   STATUS[376].EXT.AckRequired := FALSE;
   STATUS[376].EXT.Maintanence := FALSE;
   STATUS[376].EXT.Operation := FALSE;
   STATUS[376].EXT.Forced := FALSE;
   STATUS[376].EXT.BIT29 := FALSE;
   STATUS[376].EXT.BIT30 := FALSE;
   STATUS[376].EXT.BIT31 := FALSE;
   STATUS[376].EXT.ModeBit1 := FALSE;
   STATUS[376].EXT.ModeBit2 := FALSE;
   STATUS[376].EXT.ModeBit3 := FALSE;
   STATUS[376].EXT.BIT19 := FALSE;
   STATUS[376].EXT.BIT20 := FALSE;
   STATUS[376].EXT.AlarmSuppressed := FALSE;
   STATUS[376].EXT.AlarmPresent := FALSE;
   STATUS[376].EXT.AlarmFailUnAck := FALSE;
   STATUS[376].Status := 0;
   STATUS[376].TimeStamp := 16#0000;
   STATUS[377].EXT.AlarmWarnUnAck := FALSE;
   STATUS[377].EXT.AckRequired := FALSE;
   STATUS[377].EXT.Maintanence := FALSE;
   STATUS[377].EXT.Operation := FALSE;
   STATUS[377].EXT.Forced := FALSE;
   STATUS[377].EXT.BIT29 := FALSE;
   STATUS[377].EXT.BIT30 := FALSE;
   STATUS[377].EXT.BIT31 := FALSE;
   STATUS[377].EXT.ModeBit1 := FALSE;
   STATUS[377].EXT.ModeBit2 := FALSE;
   STATUS[377].EXT.ModeBit3 := FALSE;
   STATUS[377].EXT.BIT19 := FALSE;
   STATUS[377].EXT.BIT20 := FALSE;
   STATUS[377].EXT.AlarmSuppressed := FALSE;
   STATUS[377].EXT.AlarmPresent := FALSE;
   STATUS[377].EXT.AlarmFailUnAck := FALSE;
   STATUS[377].Status := 0;
   STATUS[377].TimeStamp := 16#0000;
   STATUS[378].EXT.AlarmWarnUnAck := FALSE;
   STATUS[378].EXT.AckRequired := FALSE;
   STATUS[378].EXT.Maintanence := FALSE;
   STATUS[378].EXT.Operation := FALSE;
   STATUS[378].EXT.Forced := FALSE;
   STATUS[378].EXT.BIT29 := FALSE;
   STATUS[378].EXT.BIT30 := FALSE;
   STATUS[378].EXT.BIT31 := FALSE;
   STATUS[378].EXT.ModeBit1 := FALSE;
   STATUS[378].EXT.ModeBit2 := FALSE;
   STATUS[378].EXT.ModeBit3 := FALSE;
   STATUS[378].EXT.BIT19 := FALSE;
   STATUS[378].EXT.BIT20 := FALSE;
   STATUS[378].EXT.AlarmSuppressed := FALSE;
   STATUS[378].EXT.AlarmPresent := FALSE;
   STATUS[378].EXT.AlarmFailUnAck := FALSE;
   STATUS[378].Status := 0;
   STATUS[378].TimeStamp := 16#0000;
   STATUS[379].EXT.AlarmWarnUnAck := FALSE;
   STATUS[379].EXT.AckRequired := FALSE;
   STATUS[379].EXT.Maintanence := FALSE;
   STATUS[379].EXT.Operation := FALSE;
   STATUS[379].EXT.Forced := FALSE;
   STATUS[379].EXT.BIT29 := FALSE;
   STATUS[379].EXT.BIT30 := FALSE;
   STATUS[379].EXT.BIT31 := FALSE;
   STATUS[379].EXT.ModeBit1 := FALSE;
   STATUS[379].EXT.ModeBit2 := FALSE;
   STATUS[379].EXT.ModeBit3 := FALSE;
   STATUS[379].EXT.BIT19 := FALSE;
   STATUS[379].EXT.BIT20 := FALSE;
   STATUS[379].EXT.AlarmSuppressed := FALSE;
   STATUS[379].EXT.AlarmPresent := FALSE;
   STATUS[379].EXT.AlarmFailUnAck := FALSE;
   STATUS[379].Status := 0;
   STATUS[379].TimeStamp := 16#0000;
   STATUS[380].EXT.AlarmWarnUnAck := FALSE;
   STATUS[380].EXT.AckRequired := FALSE;
   STATUS[380].EXT.Maintanence := FALSE;
   STATUS[380].EXT.Operation := FALSE;
   STATUS[380].EXT.Forced := FALSE;
   STATUS[380].EXT.BIT29 := FALSE;
   STATUS[380].EXT.BIT30 := FALSE;
   STATUS[380].EXT.BIT31 := FALSE;
   STATUS[380].EXT.ModeBit1 := FALSE;
   STATUS[380].EXT.ModeBit2 := FALSE;
   STATUS[380].EXT.ModeBit3 := FALSE;
   STATUS[380].EXT.BIT19 := FALSE;
   STATUS[380].EXT.BIT20 := FALSE;
   STATUS[380].EXT.AlarmSuppressed := FALSE;
   STATUS[380].EXT.AlarmPresent := FALSE;
   STATUS[380].EXT.AlarmFailUnAck := FALSE;
   STATUS[380].Status := 0;
   STATUS[380].TimeStamp := 16#0000;
   STATUS[381].EXT.AlarmWarnUnAck := FALSE;
   STATUS[381].EXT.AckRequired := FALSE;
   STATUS[381].EXT.Maintanence := FALSE;
   STATUS[381].EXT.Operation := FALSE;
   STATUS[381].EXT.Forced := FALSE;
   STATUS[381].EXT.BIT29 := FALSE;
   STATUS[381].EXT.BIT30 := FALSE;
   STATUS[381].EXT.BIT31 := FALSE;
   STATUS[381].EXT.ModeBit1 := FALSE;
   STATUS[381].EXT.ModeBit2 := FALSE;
   STATUS[381].EXT.ModeBit3 := FALSE;
   STATUS[381].EXT.BIT19 := FALSE;
   STATUS[381].EXT.BIT20 := FALSE;
   STATUS[381].EXT.AlarmSuppressed := FALSE;
   STATUS[381].EXT.AlarmPresent := FALSE;
   STATUS[381].EXT.AlarmFailUnAck := FALSE;
   STATUS[381].Status := 0;
   STATUS[381].TimeStamp := 16#0000;
   STATUS[382].EXT.AlarmWarnUnAck := FALSE;
   STATUS[382].EXT.AckRequired := FALSE;
   STATUS[382].EXT.Maintanence := FALSE;
   STATUS[382].EXT.Operation := FALSE;
   STATUS[382].EXT.Forced := FALSE;
   STATUS[382].EXT.BIT29 := FALSE;
   STATUS[382].EXT.BIT30 := FALSE;
   STATUS[382].EXT.BIT31 := FALSE;
   STATUS[382].EXT.ModeBit1 := FALSE;
   STATUS[382].EXT.ModeBit2 := FALSE;
   STATUS[382].EXT.ModeBit3 := FALSE;
   STATUS[382].EXT.BIT19 := FALSE;
   STATUS[382].EXT.BIT20 := FALSE;
   STATUS[382].EXT.AlarmSuppressed := FALSE;
   STATUS[382].EXT.AlarmPresent := FALSE;
   STATUS[382].EXT.AlarmFailUnAck := FALSE;
   STATUS[382].Status := 0;
   STATUS[382].TimeStamp := 16#0000;
   STATUS[383].EXT.AlarmWarnUnAck := FALSE;
   STATUS[383].EXT.AckRequired := FALSE;
   STATUS[383].EXT.Maintanence := FALSE;
   STATUS[383].EXT.Operation := FALSE;
   STATUS[383].EXT.Forced := FALSE;
   STATUS[383].EXT.BIT29 := FALSE;
   STATUS[383].EXT.BIT30 := FALSE;
   STATUS[383].EXT.BIT31 := FALSE;
   STATUS[383].EXT.ModeBit1 := FALSE;
   STATUS[383].EXT.ModeBit2 := FALSE;
   STATUS[383].EXT.ModeBit3 := FALSE;
   STATUS[383].EXT.BIT19 := FALSE;
   STATUS[383].EXT.BIT20 := FALSE;
   STATUS[383].EXT.AlarmSuppressed := FALSE;
   STATUS[383].EXT.AlarmPresent := FALSE;
   STATUS[383].EXT.AlarmFailUnAck := FALSE;
   STATUS[383].Status := 0;
   STATUS[383].TimeStamp := 16#0000;
   STATUS[384].EXT.AlarmWarnUnAck := FALSE;
   STATUS[384].EXT.AckRequired := FALSE;
   STATUS[384].EXT.Maintanence := FALSE;
   STATUS[384].EXT.Operation := FALSE;
   STATUS[384].EXT.Forced := FALSE;
   STATUS[384].EXT.BIT29 := FALSE;
   STATUS[384].EXT.BIT30 := FALSE;
   STATUS[384].EXT.BIT31 := FALSE;
   STATUS[384].EXT.ModeBit1 := FALSE;
   STATUS[384].EXT.ModeBit2 := FALSE;
   STATUS[384].EXT.ModeBit3 := FALSE;
   STATUS[384].EXT.BIT19 := FALSE;
   STATUS[384].EXT.BIT20 := FALSE;
   STATUS[384].EXT.AlarmSuppressed := FALSE;
   STATUS[384].EXT.AlarmPresent := FALSE;
   STATUS[384].EXT.AlarmFailUnAck := FALSE;
   STATUS[384].Status := 0;
   STATUS[384].TimeStamp := 16#0000;
   STATUS[385].EXT.AlarmWarnUnAck := FALSE;
   STATUS[385].EXT.AckRequired := FALSE;
   STATUS[385].EXT.Maintanence := FALSE;
   STATUS[385].EXT.Operation := FALSE;
   STATUS[385].EXT.Forced := FALSE;
   STATUS[385].EXT.BIT29 := FALSE;
   STATUS[385].EXT.BIT30 := FALSE;
   STATUS[385].EXT.BIT31 := FALSE;
   STATUS[385].EXT.ModeBit1 := FALSE;
   STATUS[385].EXT.ModeBit2 := FALSE;
   STATUS[385].EXT.ModeBit3 := FALSE;
   STATUS[385].EXT.BIT19 := FALSE;
   STATUS[385].EXT.BIT20 := FALSE;
   STATUS[385].EXT.AlarmSuppressed := FALSE;
   STATUS[385].EXT.AlarmPresent := FALSE;
   STATUS[385].EXT.AlarmFailUnAck := FALSE;
   STATUS[385].Status := 0;
   STATUS[385].TimeStamp := 16#0000;
   STATUS[386].EXT.AlarmWarnUnAck := FALSE;
   STATUS[386].EXT.AckRequired := FALSE;
   STATUS[386].EXT.Maintanence := FALSE;
   STATUS[386].EXT.Operation := FALSE;
   STATUS[386].EXT.Forced := FALSE;
   STATUS[386].EXT.BIT29 := FALSE;
   STATUS[386].EXT.BIT30 := FALSE;
   STATUS[386].EXT.BIT31 := FALSE;
   STATUS[386].EXT.ModeBit1 := FALSE;
   STATUS[386].EXT.ModeBit2 := FALSE;
   STATUS[386].EXT.ModeBit3 := FALSE;
   STATUS[386].EXT.BIT19 := FALSE;
   STATUS[386].EXT.BIT20 := FALSE;
   STATUS[386].EXT.AlarmSuppressed := FALSE;
   STATUS[386].EXT.AlarmPresent := FALSE;
   STATUS[386].EXT.AlarmFailUnAck := FALSE;
   STATUS[386].Status := 0;
   STATUS[386].TimeStamp := 16#0000;
   STATUS[387].EXT.AlarmWarnUnAck := FALSE;
   STATUS[387].EXT.AckRequired := FALSE;
   STATUS[387].EXT.Maintanence := FALSE;
   STATUS[387].EXT.Operation := FALSE;
   STATUS[387].EXT.Forced := FALSE;
   STATUS[387].EXT.BIT29 := FALSE;
   STATUS[387].EXT.BIT30 := FALSE;
   STATUS[387].EXT.BIT31 := FALSE;
   STATUS[387].EXT.ModeBit1 := FALSE;
   STATUS[387].EXT.ModeBit2 := FALSE;
   STATUS[387].EXT.ModeBit3 := FALSE;
   STATUS[387].EXT.BIT19 := FALSE;
   STATUS[387].EXT.BIT20 := FALSE;
   STATUS[387].EXT.AlarmSuppressed := FALSE;
   STATUS[387].EXT.AlarmPresent := FALSE;
   STATUS[387].EXT.AlarmFailUnAck := FALSE;
   STATUS[387].Status := 0;
   STATUS[387].TimeStamp := 16#0000;
   STATUS[388].EXT.AlarmWarnUnAck := FALSE;
   STATUS[388].EXT.AckRequired := FALSE;
   STATUS[388].EXT.Maintanence := FALSE;
   STATUS[388].EXT.Operation := FALSE;
   STATUS[388].EXT.Forced := FALSE;
   STATUS[388].EXT.BIT29 := FALSE;
   STATUS[388].EXT.BIT30 := FALSE;
   STATUS[388].EXT.BIT31 := FALSE;
   STATUS[388].EXT.ModeBit1 := FALSE;
   STATUS[388].EXT.ModeBit2 := FALSE;
   STATUS[388].EXT.ModeBit3 := FALSE;
   STATUS[388].EXT.BIT19 := FALSE;
   STATUS[388].EXT.BIT20 := FALSE;
   STATUS[388].EXT.AlarmSuppressed := FALSE;
   STATUS[388].EXT.AlarmPresent := FALSE;
   STATUS[388].EXT.AlarmFailUnAck := FALSE;
   STATUS[388].Status := 0;
   STATUS[388].TimeStamp := 16#0000;
   STATUS[389].EXT.AlarmWarnUnAck := FALSE;
   STATUS[389].EXT.AckRequired := FALSE;
   STATUS[389].EXT.Maintanence := FALSE;
   STATUS[389].EXT.Operation := FALSE;
   STATUS[389].EXT.Forced := FALSE;
   STATUS[389].EXT.BIT29 := FALSE;
   STATUS[389].EXT.BIT30 := FALSE;
   STATUS[389].EXT.BIT31 := FALSE;
   STATUS[389].EXT.ModeBit1 := FALSE;
   STATUS[389].EXT.ModeBit2 := FALSE;
   STATUS[389].EXT.ModeBit3 := FALSE;
   STATUS[389].EXT.BIT19 := FALSE;
   STATUS[389].EXT.BIT20 := FALSE;
   STATUS[389].EXT.AlarmSuppressed := FALSE;
   STATUS[389].EXT.AlarmPresent := FALSE;
   STATUS[389].EXT.AlarmFailUnAck := FALSE;
   STATUS[389].Status := 0;
   STATUS[389].TimeStamp := 16#0000;
   STATUS[390].EXT.AlarmWarnUnAck := FALSE;
   STATUS[390].EXT.AckRequired := FALSE;
   STATUS[390].EXT.Maintanence := FALSE;
   STATUS[390].EXT.Operation := FALSE;
   STATUS[390].EXT.Forced := FALSE;
   STATUS[390].EXT.BIT29 := FALSE;
   STATUS[390].EXT.BIT30 := FALSE;
   STATUS[390].EXT.BIT31 := FALSE;
   STATUS[390].EXT.ModeBit1 := FALSE;
   STATUS[390].EXT.ModeBit2 := FALSE;
   STATUS[390].EXT.ModeBit3 := FALSE;
   STATUS[390].EXT.BIT19 := FALSE;
   STATUS[390].EXT.BIT20 := FALSE;
   STATUS[390].EXT.AlarmSuppressed := FALSE;
   STATUS[390].EXT.AlarmPresent := FALSE;
   STATUS[390].EXT.AlarmFailUnAck := FALSE;
   STATUS[390].Status := 0;
   STATUS[390].TimeStamp := 16#0000;
   STATUS[391].EXT.AlarmWarnUnAck := FALSE;
   STATUS[391].EXT.AckRequired := FALSE;
   STATUS[391].EXT.Maintanence := FALSE;
   STATUS[391].EXT.Operation := FALSE;
   STATUS[391].EXT.Forced := FALSE;
   STATUS[391].EXT.BIT29 := FALSE;
   STATUS[391].EXT.BIT30 := FALSE;
   STATUS[391].EXT.BIT31 := FALSE;
   STATUS[391].EXT.ModeBit1 := FALSE;
   STATUS[391].EXT.ModeBit2 := FALSE;
   STATUS[391].EXT.ModeBit3 := FALSE;
   STATUS[391].EXT.BIT19 := FALSE;
   STATUS[391].EXT.BIT20 := FALSE;
   STATUS[391].EXT.AlarmSuppressed := FALSE;
   STATUS[391].EXT.AlarmPresent := FALSE;
   STATUS[391].EXT.AlarmFailUnAck := FALSE;
   STATUS[391].Status := 0;
   STATUS[391].TimeStamp := 16#0000;
   STATUS[392].EXT.AlarmWarnUnAck := FALSE;
   STATUS[392].EXT.AckRequired := FALSE;
   STATUS[392].EXT.Maintanence := FALSE;
   STATUS[392].EXT.Operation := FALSE;
   STATUS[392].EXT.Forced := FALSE;
   STATUS[392].EXT.BIT29 := FALSE;
   STATUS[392].EXT.BIT30 := FALSE;
   STATUS[392].EXT.BIT31 := FALSE;
   STATUS[392].EXT.ModeBit1 := FALSE;
   STATUS[392].EXT.ModeBit2 := FALSE;
   STATUS[392].EXT.ModeBit3 := FALSE;
   STATUS[392].EXT.BIT19 := FALSE;
   STATUS[392].EXT.BIT20 := FALSE;
   STATUS[392].EXT.AlarmSuppressed := FALSE;
   STATUS[392].EXT.AlarmPresent := FALSE;
   STATUS[392].EXT.AlarmFailUnAck := FALSE;
   STATUS[392].Status := 0;
   STATUS[392].TimeStamp := 16#0000;
   STATUS[393].EXT.AlarmWarnUnAck := FALSE;
   STATUS[393].EXT.AckRequired := FALSE;
   STATUS[393].EXT.Maintanence := FALSE;
   STATUS[393].EXT.Operation := FALSE;
   STATUS[393].EXT.Forced := FALSE;
   STATUS[393].EXT.BIT29 := FALSE;
   STATUS[393].EXT.BIT30 := FALSE;
   STATUS[393].EXT.BIT31 := FALSE;
   STATUS[393].EXT.ModeBit1 := FALSE;
   STATUS[393].EXT.ModeBit2 := FALSE;
   STATUS[393].EXT.ModeBit3 := FALSE;
   STATUS[393].EXT.BIT19 := FALSE;
   STATUS[393].EXT.BIT20 := FALSE;
   STATUS[393].EXT.AlarmSuppressed := FALSE;
   STATUS[393].EXT.AlarmPresent := FALSE;
   STATUS[393].EXT.AlarmFailUnAck := FALSE;
   STATUS[393].Status := 0;
   STATUS[393].TimeStamp := 16#0000;
   STATUS[394].EXT.AlarmWarnUnAck := FALSE;
   STATUS[394].EXT.AckRequired := FALSE;
   STATUS[394].EXT.Maintanence := FALSE;
   STATUS[394].EXT.Operation := FALSE;
   STATUS[394].EXT.Forced := FALSE;
   STATUS[394].EXT.BIT29 := FALSE;
   STATUS[394].EXT.BIT30 := FALSE;
   STATUS[394].EXT.BIT31 := FALSE;
   STATUS[394].EXT.ModeBit1 := FALSE;
   STATUS[394].EXT.ModeBit2 := FALSE;
   STATUS[394].EXT.ModeBit3 := FALSE;
   STATUS[394].EXT.BIT19 := FALSE;
   STATUS[394].EXT.BIT20 := FALSE;
   STATUS[394].EXT.AlarmSuppressed := FALSE;
   STATUS[394].EXT.AlarmPresent := FALSE;
   STATUS[394].EXT.AlarmFailUnAck := FALSE;
   STATUS[394].Status := 0;
   STATUS[394].TimeStamp := 16#0000;
   STATUS[395].EXT.AlarmWarnUnAck := FALSE;
   STATUS[395].EXT.AckRequired := FALSE;
   STATUS[395].EXT.Maintanence := FALSE;
   STATUS[395].EXT.Operation := FALSE;
   STATUS[395].EXT.Forced := FALSE;
   STATUS[395].EXT.BIT29 := FALSE;
   STATUS[395].EXT.BIT30 := FALSE;
   STATUS[395].EXT.BIT31 := FALSE;
   STATUS[395].EXT.ModeBit1 := FALSE;
   STATUS[395].EXT.ModeBit2 := FALSE;
   STATUS[395].EXT.ModeBit3 := FALSE;
   STATUS[395].EXT.BIT19 := FALSE;
   STATUS[395].EXT.BIT20 := FALSE;
   STATUS[395].EXT.AlarmSuppressed := FALSE;
   STATUS[395].EXT.AlarmPresent := FALSE;
   STATUS[395].EXT.AlarmFailUnAck := FALSE;
   STATUS[395].Status := 0;
   STATUS[395].TimeStamp := 16#0000;
   STATUS[396].EXT.AlarmWarnUnAck := FALSE;
   STATUS[396].EXT.AckRequired := FALSE;
   STATUS[396].EXT.Maintanence := FALSE;
   STATUS[396].EXT.Operation := FALSE;
   STATUS[396].EXT.Forced := FALSE;
   STATUS[396].EXT.BIT29 := FALSE;
   STATUS[396].EXT.BIT30 := FALSE;
   STATUS[396].EXT.BIT31 := FALSE;
   STATUS[396].EXT.ModeBit1 := FALSE;
   STATUS[396].EXT.ModeBit2 := FALSE;
   STATUS[396].EXT.ModeBit3 := FALSE;
   STATUS[396].EXT.BIT19 := FALSE;
   STATUS[396].EXT.BIT20 := FALSE;
   STATUS[396].EXT.AlarmSuppressed := FALSE;
   STATUS[396].EXT.AlarmPresent := FALSE;
   STATUS[396].EXT.AlarmFailUnAck := FALSE;
   STATUS[396].Status := 0;
   STATUS[396].TimeStamp := 16#0000;
   STATUS[397].EXT.AlarmWarnUnAck := FALSE;
   STATUS[397].EXT.AckRequired := FALSE;
   STATUS[397].EXT.Maintanence := FALSE;
   STATUS[397].EXT.Operation := FALSE;
   STATUS[397].EXT.Forced := FALSE;
   STATUS[397].EXT.BIT29 := FALSE;
   STATUS[397].EXT.BIT30 := FALSE;
   STATUS[397].EXT.BIT31 := FALSE;
   STATUS[397].EXT.ModeBit1 := FALSE;
   STATUS[397].EXT.ModeBit2 := FALSE;
   STATUS[397].EXT.ModeBit3 := FALSE;
   STATUS[397].EXT.BIT19 := FALSE;
   STATUS[397].EXT.BIT20 := FALSE;
   STATUS[397].EXT.AlarmSuppressed := FALSE;
   STATUS[397].EXT.AlarmPresent := FALSE;
   STATUS[397].EXT.AlarmFailUnAck := FALSE;
   STATUS[397].Status := 0;
   STATUS[397].TimeStamp := 16#0000;
   STATUS[398].EXT.AlarmWarnUnAck := FALSE;
   STATUS[398].EXT.AckRequired := FALSE;
   STATUS[398].EXT.Maintanence := FALSE;
   STATUS[398].EXT.Operation := FALSE;
   STATUS[398].EXT.Forced := FALSE;
   STATUS[398].EXT.BIT29 := FALSE;
   STATUS[398].EXT.BIT30 := FALSE;
   STATUS[398].EXT.BIT31 := FALSE;
   STATUS[398].EXT.ModeBit1 := FALSE;
   STATUS[398].EXT.ModeBit2 := FALSE;
   STATUS[398].EXT.ModeBit3 := FALSE;
   STATUS[398].EXT.BIT19 := FALSE;
   STATUS[398].EXT.BIT20 := FALSE;
   STATUS[398].EXT.AlarmSuppressed := FALSE;
   STATUS[398].EXT.AlarmPresent := FALSE;
   STATUS[398].EXT.AlarmFailUnAck := FALSE;
   STATUS[398].Status := 0;
   STATUS[398].TimeStamp := 16#0000;
   STATUS[399].EXT.AlarmWarnUnAck := FALSE;
   STATUS[399].EXT.AckRequired := FALSE;
   STATUS[399].EXT.Maintanence := FALSE;
   STATUS[399].EXT.Operation := FALSE;
   STATUS[399].EXT.Forced := FALSE;
   STATUS[399].EXT.BIT29 := FALSE;
   STATUS[399].EXT.BIT30 := FALSE;
   STATUS[399].EXT.BIT31 := FALSE;
   STATUS[399].EXT.ModeBit1 := FALSE;
   STATUS[399].EXT.ModeBit2 := FALSE;
   STATUS[399].EXT.ModeBit3 := FALSE;
   STATUS[399].EXT.BIT19 := FALSE;
   STATUS[399].EXT.BIT20 := FALSE;
   STATUS[399].EXT.AlarmSuppressed := FALSE;
   STATUS[399].EXT.AlarmPresent := FALSE;
   STATUS[399].EXT.AlarmFailUnAck := FALSE;
   STATUS[399].Status := 0;
   STATUS[399].TimeStamp := 16#0000;
   STATUS[400].EXT.AlarmWarnUnAck := FALSE;
   STATUS[400].EXT.AckRequired := FALSE;
   STATUS[400].EXT.Maintanence := FALSE;
   STATUS[400].EXT.Operation := FALSE;
   STATUS[400].EXT.Forced := FALSE;
   STATUS[400].EXT.BIT29 := FALSE;
   STATUS[400].EXT.BIT30 := FALSE;
   STATUS[400].EXT.BIT31 := FALSE;
   STATUS[400].EXT.ModeBit1 := FALSE;
   STATUS[400].EXT.ModeBit2 := FALSE;
   STATUS[400].EXT.ModeBit3 := FALSE;
   STATUS[400].EXT.BIT19 := FALSE;
   STATUS[400].EXT.BIT20 := FALSE;
   STATUS[400].EXT.AlarmSuppressed := FALSE;
   STATUS[400].EXT.AlarmPresent := FALSE;
   STATUS[400].EXT.AlarmFailUnAck := FALSE;
   STATUS[400].Status := 0;
   STATUS[400].TimeStamp := 16#0000;
   STATUS[401].EXT.AlarmWarnUnAck := FALSE;
   STATUS[401].EXT.AckRequired := FALSE;
   STATUS[401].EXT.Maintanence := FALSE;
   STATUS[401].EXT.Operation := FALSE;
   STATUS[401].EXT.Forced := FALSE;
   STATUS[401].EXT.BIT29 := FALSE;
   STATUS[401].EXT.BIT30 := FALSE;
   STATUS[401].EXT.BIT31 := FALSE;
   STATUS[401].EXT.ModeBit1 := FALSE;
   STATUS[401].EXT.ModeBit2 := FALSE;
   STATUS[401].EXT.ModeBit3 := FALSE;
   STATUS[401].EXT.BIT19 := FALSE;
   STATUS[401].EXT.BIT20 := FALSE;
   STATUS[401].EXT.AlarmSuppressed := FALSE;
   STATUS[401].EXT.AlarmPresent := FALSE;
   STATUS[401].EXT.AlarmFailUnAck := FALSE;
   STATUS[401].Status := 0;
   STATUS[401].TimeStamp := 16#0000;
   STATUS[402].EXT.AlarmWarnUnAck := FALSE;
   STATUS[402].EXT.AckRequired := FALSE;
   STATUS[402].EXT.Maintanence := FALSE;
   STATUS[402].EXT.Operation := FALSE;
   STATUS[402].EXT.Forced := FALSE;
   STATUS[402].EXT.BIT29 := FALSE;
   STATUS[402].EXT.BIT30 := FALSE;
   STATUS[402].EXT.BIT31 := FALSE;
   STATUS[402].EXT.ModeBit1 := FALSE;
   STATUS[402].EXT.ModeBit2 := FALSE;
   STATUS[402].EXT.ModeBit3 := FALSE;
   STATUS[402].EXT.BIT19 := FALSE;
   STATUS[402].EXT.BIT20 := FALSE;
   STATUS[402].EXT.AlarmSuppressed := FALSE;
   STATUS[402].EXT.AlarmPresent := FALSE;
   STATUS[402].EXT.AlarmFailUnAck := FALSE;
   STATUS[402].Status := 0;
   STATUS[402].TimeStamp := 16#0000;
   STATUS[403].EXT.AlarmWarnUnAck := FALSE;
   STATUS[403].EXT.AckRequired := FALSE;
   STATUS[403].EXT.Maintanence := FALSE;
   STATUS[403].EXT.Operation := FALSE;
   STATUS[403].EXT.Forced := FALSE;
   STATUS[403].EXT.BIT29 := FALSE;
   STATUS[403].EXT.BIT30 := FALSE;
   STATUS[403].EXT.BIT31 := FALSE;
   STATUS[403].EXT.ModeBit1 := FALSE;
   STATUS[403].EXT.ModeBit2 := FALSE;
   STATUS[403].EXT.ModeBit3 := FALSE;
   STATUS[403].EXT.BIT19 := FALSE;
   STATUS[403].EXT.BIT20 := FALSE;
   STATUS[403].EXT.AlarmSuppressed := FALSE;
   STATUS[403].EXT.AlarmPresent := FALSE;
   STATUS[403].EXT.AlarmFailUnAck := FALSE;
   STATUS[403].Status := 0;
   STATUS[403].TimeStamp := 16#0000;
   STATUS[404].EXT.AlarmWarnUnAck := FALSE;
   STATUS[404].EXT.AckRequired := FALSE;
   STATUS[404].EXT.Maintanence := FALSE;
   STATUS[404].EXT.Operation := FALSE;
   STATUS[404].EXT.Forced := FALSE;
   STATUS[404].EXT.BIT29 := FALSE;
   STATUS[404].EXT.BIT30 := FALSE;
   STATUS[404].EXT.BIT31 := FALSE;
   STATUS[404].EXT.ModeBit1 := FALSE;
   STATUS[404].EXT.ModeBit2 := FALSE;
   STATUS[404].EXT.ModeBit3 := FALSE;
   STATUS[404].EXT.BIT19 := FALSE;
   STATUS[404].EXT.BIT20 := FALSE;
   STATUS[404].EXT.AlarmSuppressed := FALSE;
   STATUS[404].EXT.AlarmPresent := FALSE;
   STATUS[404].EXT.AlarmFailUnAck := FALSE;
   STATUS[404].Status := 0;
   STATUS[404].TimeStamp := 16#0000;
   STATUS[405].EXT.AlarmWarnUnAck := FALSE;
   STATUS[405].EXT.AckRequired := FALSE;
   STATUS[405].EXT.Maintanence := FALSE;
   STATUS[405].EXT.Operation := FALSE;
   STATUS[405].EXT.Forced := FALSE;
   STATUS[405].EXT.BIT29 := FALSE;
   STATUS[405].EXT.BIT30 := FALSE;
   STATUS[405].EXT.BIT31 := FALSE;
   STATUS[405].EXT.ModeBit1 := FALSE;
   STATUS[405].EXT.ModeBit2 := FALSE;
   STATUS[405].EXT.ModeBit3 := FALSE;
   STATUS[405].EXT.BIT19 := FALSE;
   STATUS[405].EXT.BIT20 := FALSE;
   STATUS[405].EXT.AlarmSuppressed := FALSE;
   STATUS[405].EXT.AlarmPresent := FALSE;
   STATUS[405].EXT.AlarmFailUnAck := FALSE;
   STATUS[405].Status := 0;
   STATUS[405].TimeStamp := 16#0000;
   STATUS[406].EXT.AlarmWarnUnAck := FALSE;
   STATUS[406].EXT.AckRequired := FALSE;
   STATUS[406].EXT.Maintanence := FALSE;
   STATUS[406].EXT.Operation := FALSE;
   STATUS[406].EXT.Forced := FALSE;
   STATUS[406].EXT.BIT29 := FALSE;
   STATUS[406].EXT.BIT30 := FALSE;
   STATUS[406].EXT.BIT31 := FALSE;
   STATUS[406].EXT.ModeBit1 := FALSE;
   STATUS[406].EXT.ModeBit2 := FALSE;
   STATUS[406].EXT.ModeBit3 := FALSE;
   STATUS[406].EXT.BIT19 := FALSE;
   STATUS[406].EXT.BIT20 := FALSE;
   STATUS[406].EXT.AlarmSuppressed := FALSE;
   STATUS[406].EXT.AlarmPresent := FALSE;
   STATUS[406].EXT.AlarmFailUnAck := FALSE;
   STATUS[406].Status := 0;
   STATUS[406].TimeStamp := 16#0000;
   STATUS[407].EXT.AlarmWarnUnAck := FALSE;
   STATUS[407].EXT.AckRequired := FALSE;
   STATUS[407].EXT.Maintanence := FALSE;
   STATUS[407].EXT.Operation := FALSE;
   STATUS[407].EXT.Forced := FALSE;
   STATUS[407].EXT.BIT29 := FALSE;
   STATUS[407].EXT.BIT30 := FALSE;
   STATUS[407].EXT.BIT31 := FALSE;
   STATUS[407].EXT.ModeBit1 := FALSE;
   STATUS[407].EXT.ModeBit2 := FALSE;
   STATUS[407].EXT.ModeBit3 := FALSE;
   STATUS[407].EXT.BIT19 := FALSE;
   STATUS[407].EXT.BIT20 := FALSE;
   STATUS[407].EXT.AlarmSuppressed := FALSE;
   STATUS[407].EXT.AlarmPresent := FALSE;
   STATUS[407].EXT.AlarmFailUnAck := FALSE;
   STATUS[407].Status := 0;
   STATUS[407].TimeStamp := 16#0000;
   STATUS[408].EXT.AlarmWarnUnAck := FALSE;
   STATUS[408].EXT.AckRequired := FALSE;
   STATUS[408].EXT.Maintanence := FALSE;
   STATUS[408].EXT.Operation := FALSE;
   STATUS[408].EXT.Forced := FALSE;
   STATUS[408].EXT.BIT29 := FALSE;
   STATUS[408].EXT.BIT30 := FALSE;
   STATUS[408].EXT.BIT31 := FALSE;
   STATUS[408].EXT.ModeBit1 := FALSE;
   STATUS[408].EXT.ModeBit2 := FALSE;
   STATUS[408].EXT.ModeBit3 := FALSE;
   STATUS[408].EXT.BIT19 := FALSE;
   STATUS[408].EXT.BIT20 := FALSE;
   STATUS[408].EXT.AlarmSuppressed := FALSE;
   STATUS[408].EXT.AlarmPresent := FALSE;
   STATUS[408].EXT.AlarmFailUnAck := FALSE;
   STATUS[408].Status := 0;
   STATUS[408].TimeStamp := 16#0000;
   STATUS[409].EXT.AlarmWarnUnAck := FALSE;
   STATUS[409].EXT.AckRequired := FALSE;
   STATUS[409].EXT.Maintanence := FALSE;
   STATUS[409].EXT.Operation := FALSE;
   STATUS[409].EXT.Forced := FALSE;
   STATUS[409].EXT.BIT29 := FALSE;
   STATUS[409].EXT.BIT30 := FALSE;
   STATUS[409].EXT.BIT31 := FALSE;
   STATUS[409].EXT.ModeBit1 := FALSE;
   STATUS[409].EXT.ModeBit2 := FALSE;
   STATUS[409].EXT.ModeBit3 := FALSE;
   STATUS[409].EXT.BIT19 := FALSE;
   STATUS[409].EXT.BIT20 := FALSE;
   STATUS[409].EXT.AlarmSuppressed := FALSE;
   STATUS[409].EXT.AlarmPresent := FALSE;
   STATUS[409].EXT.AlarmFailUnAck := FALSE;
   STATUS[409].Status := 0;
   STATUS[409].TimeStamp := 16#0000;
   STATUS[410].EXT.AlarmWarnUnAck := FALSE;
   STATUS[410].EXT.AckRequired := FALSE;
   STATUS[410].EXT.Maintanence := FALSE;
   STATUS[410].EXT.Operation := FALSE;
   STATUS[410].EXT.Forced := FALSE;
   STATUS[410].EXT.BIT29 := FALSE;
   STATUS[410].EXT.BIT30 := FALSE;
   STATUS[410].EXT.BIT31 := FALSE;
   STATUS[410].EXT.ModeBit1 := FALSE;
   STATUS[410].EXT.ModeBit2 := FALSE;
   STATUS[410].EXT.ModeBit3 := FALSE;
   STATUS[410].EXT.BIT19 := FALSE;
   STATUS[410].EXT.BIT20 := FALSE;
   STATUS[410].EXT.AlarmSuppressed := FALSE;
   STATUS[410].EXT.AlarmPresent := FALSE;
   STATUS[410].EXT.AlarmFailUnAck := FALSE;
   STATUS[410].Status := 0;
   STATUS[410].TimeStamp := 16#0000;
   STATUS[411].EXT.AlarmWarnUnAck := FALSE;
   STATUS[411].EXT.AckRequired := FALSE;
   STATUS[411].EXT.Maintanence := FALSE;
   STATUS[411].EXT.Operation := FALSE;
   STATUS[411].EXT.Forced := FALSE;
   STATUS[411].EXT.BIT29 := FALSE;
   STATUS[411].EXT.BIT30 := FALSE;
   STATUS[411].EXT.BIT31 := FALSE;
   STATUS[411].EXT.ModeBit1 := FALSE;
   STATUS[411].EXT.ModeBit2 := FALSE;
   STATUS[411].EXT.ModeBit3 := FALSE;
   STATUS[411].EXT.BIT19 := FALSE;
   STATUS[411].EXT.BIT20 := FALSE;
   STATUS[411].EXT.AlarmSuppressed := FALSE;
   STATUS[411].EXT.AlarmPresent := FALSE;
   STATUS[411].EXT.AlarmFailUnAck := FALSE;
   STATUS[411].Status := 0;
   STATUS[411].TimeStamp := 16#0000;
   STATUS[412].EXT.AlarmWarnUnAck := FALSE;
   STATUS[412].EXT.AckRequired := FALSE;
   STATUS[412].EXT.Maintanence := FALSE;
   STATUS[412].EXT.Operation := FALSE;
   STATUS[412].EXT.Forced := FALSE;
   STATUS[412].EXT.BIT29 := FALSE;
   STATUS[412].EXT.BIT30 := FALSE;
   STATUS[412].EXT.BIT31 := FALSE;
   STATUS[412].EXT.ModeBit1 := FALSE;
   STATUS[412].EXT.ModeBit2 := FALSE;
   STATUS[412].EXT.ModeBit3 := FALSE;
   STATUS[412].EXT.BIT19 := FALSE;
   STATUS[412].EXT.BIT20 := FALSE;
   STATUS[412].EXT.AlarmSuppressed := FALSE;
   STATUS[412].EXT.AlarmPresent := FALSE;
   STATUS[412].EXT.AlarmFailUnAck := FALSE;
   STATUS[412].Status := 0;
   STATUS[412].TimeStamp := 16#0000;
   STATUS[413].EXT.AlarmWarnUnAck := FALSE;
   STATUS[413].EXT.AckRequired := FALSE;
   STATUS[413].EXT.Maintanence := FALSE;
   STATUS[413].EXT.Operation := FALSE;
   STATUS[413].EXT.Forced := FALSE;
   STATUS[413].EXT.BIT29 := FALSE;
   STATUS[413].EXT.BIT30 := FALSE;
   STATUS[413].EXT.BIT31 := FALSE;
   STATUS[413].EXT.ModeBit1 := FALSE;
   STATUS[413].EXT.ModeBit2 := FALSE;
   STATUS[413].EXT.ModeBit3 := FALSE;
   STATUS[413].EXT.BIT19 := FALSE;
   STATUS[413].EXT.BIT20 := FALSE;
   STATUS[413].EXT.AlarmSuppressed := FALSE;
   STATUS[413].EXT.AlarmPresent := FALSE;
   STATUS[413].EXT.AlarmFailUnAck := FALSE;
   STATUS[413].Status := 0;
   STATUS[413].TimeStamp := 16#0000;
   STATUS[414].EXT.AlarmWarnUnAck := FALSE;
   STATUS[414].EXT.AckRequired := FALSE;
   STATUS[414].EXT.Maintanence := FALSE;
   STATUS[414].EXT.Operation := FALSE;
   STATUS[414].EXT.Forced := FALSE;
   STATUS[414].EXT.BIT29 := FALSE;
   STATUS[414].EXT.BIT30 := FALSE;
   STATUS[414].EXT.BIT31 := FALSE;
   STATUS[414].EXT.ModeBit1 := FALSE;
   STATUS[414].EXT.ModeBit2 := FALSE;
   STATUS[414].EXT.ModeBit3 := FALSE;
   STATUS[414].EXT.BIT19 := FALSE;
   STATUS[414].EXT.BIT20 := FALSE;
   STATUS[414].EXT.AlarmSuppressed := FALSE;
   STATUS[414].EXT.AlarmPresent := FALSE;
   STATUS[414].EXT.AlarmFailUnAck := FALSE;
   STATUS[414].Status := 0;
   STATUS[414].TimeStamp := 16#0000;
   STATUS[415].EXT.AlarmWarnUnAck := FALSE;
   STATUS[415].EXT.AckRequired := FALSE;
   STATUS[415].EXT.Maintanence := FALSE;
   STATUS[415].EXT.Operation := FALSE;
   STATUS[415].EXT.Forced := FALSE;
   STATUS[415].EXT.BIT29 := FALSE;
   STATUS[415].EXT.BIT30 := FALSE;
   STATUS[415].EXT.BIT31 := FALSE;
   STATUS[415].EXT.ModeBit1 := FALSE;
   STATUS[415].EXT.ModeBit2 := FALSE;
   STATUS[415].EXT.ModeBit3 := FALSE;
   STATUS[415].EXT.BIT19 := FALSE;
   STATUS[415].EXT.BIT20 := FALSE;
   STATUS[415].EXT.AlarmSuppressed := FALSE;
   STATUS[415].EXT.AlarmPresent := FALSE;
   STATUS[415].EXT.AlarmFailUnAck := FALSE;
   STATUS[415].Status := 0;
   STATUS[415].TimeStamp := 16#0000;
   STATUS[416].EXT.AlarmWarnUnAck := FALSE;
   STATUS[416].EXT.AckRequired := FALSE;
   STATUS[416].EXT.Maintanence := FALSE;
   STATUS[416].EXT.Operation := FALSE;
   STATUS[416].EXT.Forced := FALSE;
   STATUS[416].EXT.BIT29 := FALSE;
   STATUS[416].EXT.BIT30 := FALSE;
   STATUS[416].EXT.BIT31 := FALSE;
   STATUS[416].EXT.ModeBit1 := TRUE;
   STATUS[416].EXT.ModeBit2 := TRUE;
   STATUS[416].EXT.ModeBit3 := FALSE;
   STATUS[416].EXT.BIT19 := FALSE;
   STATUS[416].EXT.BIT20 := FALSE;
   STATUS[416].EXT.AlarmSuppressed := FALSE;
   STATUS[416].EXT.AlarmPresent := FALSE;
   STATUS[416].EXT.AlarmFailUnAck := FALSE;
   STATUS[416].Status := 1;
   STATUS[416].TimeStamp := 16#5AAD;
   STATUS[417].EXT.AlarmWarnUnAck := FALSE;
   STATUS[417].EXT.AckRequired := FALSE;
   STATUS[417].EXT.Maintanence := FALSE;
   STATUS[417].EXT.Operation := FALSE;
   STATUS[417].EXT.Forced := FALSE;
   STATUS[417].EXT.BIT29 := FALSE;
   STATUS[417].EXT.BIT30 := FALSE;
   STATUS[417].EXT.BIT31 := FALSE;
   STATUS[417].EXT.ModeBit1 := FALSE;
   STATUS[417].EXT.ModeBit2 := FALSE;
   STATUS[417].EXT.ModeBit3 := FALSE;
   STATUS[417].EXT.BIT19 := FALSE;
   STATUS[417].EXT.BIT20 := FALSE;
   STATUS[417].EXT.AlarmSuppressed := FALSE;
   STATUS[417].EXT.AlarmPresent := TRUE;
   STATUS[417].EXT.AlarmFailUnAck := TRUE;
   STATUS[417].Status := 210;
   STATUS[417].TimeStamp := 16#22AA;
   STATUS[418].EXT.AlarmWarnUnAck := FALSE;
   STATUS[418].EXT.AckRequired := FALSE;
   STATUS[418].EXT.Maintanence := FALSE;
   STATUS[418].EXT.Operation := FALSE;
   STATUS[418].EXT.Forced := FALSE;
   STATUS[418].EXT.BIT29 := FALSE;
   STATUS[418].EXT.BIT30 := FALSE;
   STATUS[418].EXT.BIT31 := FALSE;
   STATUS[418].EXT.ModeBit1 := FALSE;
   STATUS[418].EXT.ModeBit2 := FALSE;
   STATUS[418].EXT.ModeBit3 := FALSE;
   STATUS[418].EXT.BIT19 := FALSE;
   STATUS[418].EXT.BIT20 := FALSE;
   STATUS[418].EXT.AlarmSuppressed := FALSE;
   STATUS[418].EXT.AlarmPresent := FALSE;
   STATUS[418].EXT.AlarmFailUnAck := FALSE;
   STATUS[418].Status := 0;
   STATUS[418].TimeStamp := 16#0000;
   STATUS[419].EXT.AlarmWarnUnAck := FALSE;
   STATUS[419].EXT.AckRequired := FALSE;
   STATUS[419].EXT.Maintanence := FALSE;
   STATUS[419].EXT.Operation := FALSE;
   STATUS[419].EXT.Forced := FALSE;
   STATUS[419].EXT.BIT29 := FALSE;
   STATUS[419].EXT.BIT30 := FALSE;
   STATUS[419].EXT.BIT31 := FALSE;
   STATUS[419].EXT.ModeBit1 := FALSE;
   STATUS[419].EXT.ModeBit2 := FALSE;
   STATUS[419].EXT.ModeBit3 := FALSE;
   STATUS[419].EXT.BIT19 := FALSE;
   STATUS[419].EXT.BIT20 := FALSE;
   STATUS[419].EXT.AlarmSuppressed := FALSE;
   STATUS[419].EXT.AlarmPresent := FALSE;
   STATUS[419].EXT.AlarmFailUnAck := FALSE;
   STATUS[419].Status := 0;
   STATUS[419].TimeStamp := 16#0000;
   STATUS[420].EXT.AlarmWarnUnAck := FALSE;
   STATUS[420].EXT.AckRequired := FALSE;
   STATUS[420].EXT.Maintanence := FALSE;
   STATUS[420].EXT.Operation := TRUE;
   STATUS[420].EXT.Forced := FALSE;
   STATUS[420].EXT.BIT29 := FALSE;
   STATUS[420].EXT.BIT30 := FALSE;
   STATUS[420].EXT.BIT31 := FALSE;
   STATUS[420].EXT.ModeBit1 := FALSE;
   STATUS[420].EXT.ModeBit2 := TRUE;
   STATUS[420].EXT.ModeBit3 := FALSE;
   STATUS[420].EXT.BIT19 := FALSE;
   STATUS[420].EXT.BIT20 := FALSE;
   STATUS[420].EXT.AlarmSuppressed := FALSE;
   STATUS[420].EXT.AlarmPresent := FALSE;
   STATUS[420].EXT.AlarmFailUnAck := FALSE;
   STATUS[420].Status := 4177;
   STATUS[420].TimeStamp := 16#7BED;
   STATUS[421].EXT.AlarmWarnUnAck := FALSE;
   STATUS[421].EXT.AckRequired := FALSE;
   STATUS[421].EXT.Maintanence := FALSE;
   STATUS[421].EXT.Operation := FALSE;
   STATUS[421].EXT.Forced := FALSE;
   STATUS[421].EXT.BIT29 := FALSE;
   STATUS[421].EXT.BIT30 := FALSE;
   STATUS[421].EXT.BIT31 := FALSE;
   STATUS[421].EXT.ModeBit1 := FALSE;
   STATUS[421].EXT.ModeBit2 := TRUE;
   STATUS[421].EXT.ModeBit3 := FALSE;
   STATUS[421].EXT.BIT19 := FALSE;
   STATUS[421].EXT.BIT20 := FALSE;
   STATUS[421].EXT.AlarmSuppressed := FALSE;
   STATUS[421].EXT.AlarmPresent := FALSE;
   STATUS[421].EXT.AlarmFailUnAck := FALSE;
   STATUS[421].Status := 1;
   STATUS[421].TimeStamp := 16#24A4;
   STATUS[422].EXT.AlarmWarnUnAck := FALSE;
   STATUS[422].EXT.AckRequired := FALSE;
   STATUS[422].EXT.Maintanence := FALSE;
   STATUS[422].EXT.Operation := TRUE;
   STATUS[422].EXT.Forced := FALSE;
   STATUS[422].EXT.BIT29 := FALSE;
   STATUS[422].EXT.BIT30 := FALSE;
   STATUS[422].EXT.BIT31 := FALSE;
   STATUS[422].EXT.ModeBit1 := FALSE;
   STATUS[422].EXT.ModeBit2 := TRUE;
   STATUS[422].EXT.ModeBit3 := FALSE;
   STATUS[422].EXT.BIT19 := FALSE;
   STATUS[422].EXT.BIT20 := FALSE;
   STATUS[422].EXT.AlarmSuppressed := FALSE;
   STATUS[422].EXT.AlarmPresent := FALSE;
   STATUS[422].EXT.AlarmFailUnAck := FALSE;
   STATUS[422].Status := 4177;
   STATUS[422].TimeStamp := 16#88CC;
   STATUS[423].EXT.AlarmWarnUnAck := FALSE;
   STATUS[423].EXT.AckRequired := FALSE;
   STATUS[423].EXT.Maintanence := FALSE;
   STATUS[423].EXT.Operation := FALSE;
   STATUS[423].EXT.Forced := FALSE;
   STATUS[423].EXT.BIT29 := FALSE;
   STATUS[423].EXT.BIT30 := FALSE;
   STATUS[423].EXT.BIT31 := FALSE;
   STATUS[423].EXT.ModeBit1 := FALSE;
   STATUS[423].EXT.ModeBit2 := FALSE;
   STATUS[423].EXT.ModeBit3 := FALSE;
   STATUS[423].EXT.BIT19 := FALSE;
   STATUS[423].EXT.BIT20 := FALSE;
   STATUS[423].EXT.AlarmSuppressed := FALSE;
   STATUS[423].EXT.AlarmPresent := FALSE;
   STATUS[423].EXT.AlarmFailUnAck := FALSE;
   STATUS[423].Status := 1;
   STATUS[423].TimeStamp := 16#5187;
   STATUS[424].EXT.AlarmWarnUnAck := FALSE;
   STATUS[424].EXT.AckRequired := FALSE;
   STATUS[424].EXT.Maintanence := FALSE;
   STATUS[424].EXT.Operation := FALSE;
   STATUS[424].EXT.Forced := FALSE;
   STATUS[424].EXT.BIT29 := FALSE;
   STATUS[424].EXT.BIT30 := FALSE;
   STATUS[424].EXT.BIT31 := FALSE;
   STATUS[424].EXT.ModeBit1 := FALSE;
   STATUS[424].EXT.ModeBit2 := FALSE;
   STATUS[424].EXT.ModeBit3 := FALSE;
   STATUS[424].EXT.BIT19 := FALSE;
   STATUS[424].EXT.BIT20 := FALSE;
   STATUS[424].EXT.AlarmSuppressed := FALSE;
   STATUS[424].EXT.AlarmPresent := FALSE;
   STATUS[424].EXT.AlarmFailUnAck := FALSE;
   STATUS[424].Status := 0;
   STATUS[424].TimeStamp := 16#0000;
   STATUS[425].EXT.AlarmWarnUnAck := FALSE;
   STATUS[425].EXT.AckRequired := FALSE;
   STATUS[425].EXT.Maintanence := FALSE;
   STATUS[425].EXT.Operation := FALSE;
   STATUS[425].EXT.Forced := FALSE;
   STATUS[425].EXT.BIT29 := FALSE;
   STATUS[425].EXT.BIT30 := FALSE;
   STATUS[425].EXT.BIT31 := FALSE;
   STATUS[425].EXT.ModeBit1 := FALSE;
   STATUS[425].EXT.ModeBit2 := FALSE;
   STATUS[425].EXT.ModeBit3 := FALSE;
   STATUS[425].EXT.BIT19 := FALSE;
   STATUS[425].EXT.BIT20 := FALSE;
   STATUS[425].EXT.AlarmSuppressed := FALSE;
   STATUS[425].EXT.AlarmPresent := FALSE;
   STATUS[425].EXT.AlarmFailUnAck := FALSE;
   STATUS[425].Status := 0;
   STATUS[425].TimeStamp := 16#0000;
   STATUS[426].EXT.AlarmWarnUnAck := FALSE;
   STATUS[426].EXT.AckRequired := FALSE;
   STATUS[426].EXT.Maintanence := FALSE;
   STATUS[426].EXT.Operation := FALSE;
   STATUS[426].EXT.Forced := FALSE;
   STATUS[426].EXT.BIT29 := FALSE;
   STATUS[426].EXT.BIT30 := FALSE;
   STATUS[426].EXT.BIT31 := FALSE;
   STATUS[426].EXT.ModeBit1 := FALSE;
   STATUS[426].EXT.ModeBit2 := FALSE;
   STATUS[426].EXT.ModeBit3 := FALSE;
   STATUS[426].EXT.BIT19 := FALSE;
   STATUS[426].EXT.BIT20 := FALSE;
   STATUS[426].EXT.AlarmSuppressed := FALSE;
   STATUS[426].EXT.AlarmPresent := FALSE;
   STATUS[426].EXT.AlarmFailUnAck := FALSE;
   STATUS[426].Status := 0;
   STATUS[426].TimeStamp := 16#0000;
   STATUS[427].EXT.AlarmWarnUnAck := FALSE;
   STATUS[427].EXT.AckRequired := FALSE;
   STATUS[427].EXT.Maintanence := FALSE;
   STATUS[427].EXT.Operation := FALSE;
   STATUS[427].EXT.Forced := FALSE;
   STATUS[427].EXT.BIT29 := FALSE;
   STATUS[427].EXT.BIT30 := FALSE;
   STATUS[427].EXT.BIT31 := FALSE;
   STATUS[427].EXT.ModeBit1 := FALSE;
   STATUS[427].EXT.ModeBit2 := FALSE;
   STATUS[427].EXT.ModeBit3 := FALSE;
   STATUS[427].EXT.BIT19 := FALSE;
   STATUS[427].EXT.BIT20 := FALSE;
   STATUS[427].EXT.AlarmSuppressed := FALSE;
   STATUS[427].EXT.AlarmPresent := FALSE;
   STATUS[427].EXT.AlarmFailUnAck := FALSE;
   STATUS[427].Status := 0;
   STATUS[427].TimeStamp := 16#0000;
   STATUS[428].EXT.AlarmWarnUnAck := FALSE;
   STATUS[428].EXT.AckRequired := FALSE;
   STATUS[428].EXT.Maintanence := FALSE;
   STATUS[428].EXT.Operation := FALSE;
   STATUS[428].EXT.Forced := FALSE;
   STATUS[428].EXT.BIT29 := FALSE;
   STATUS[428].EXT.BIT30 := FALSE;
   STATUS[428].EXT.BIT31 := FALSE;
   STATUS[428].EXT.ModeBit1 := FALSE;
   STATUS[428].EXT.ModeBit2 := FALSE;
   STATUS[428].EXT.ModeBit3 := FALSE;
   STATUS[428].EXT.BIT19 := FALSE;
   STATUS[428].EXT.BIT20 := FALSE;
   STATUS[428].EXT.AlarmSuppressed := FALSE;
   STATUS[428].EXT.AlarmPresent := FALSE;
   STATUS[428].EXT.AlarmFailUnAck := FALSE;
   STATUS[428].Status := 0;
   STATUS[428].TimeStamp := 16#0000;
   STATUS[429].EXT.AlarmWarnUnAck := FALSE;
   STATUS[429].EXT.AckRequired := FALSE;
   STATUS[429].EXT.Maintanence := FALSE;
   STATUS[429].EXT.Operation := FALSE;
   STATUS[429].EXT.Forced := FALSE;
   STATUS[429].EXT.BIT29 := FALSE;
   STATUS[429].EXT.BIT30 := FALSE;
   STATUS[429].EXT.BIT31 := FALSE;
   STATUS[429].EXT.ModeBit1 := FALSE;
   STATUS[429].EXT.ModeBit2 := FALSE;
   STATUS[429].EXT.ModeBit3 := FALSE;
   STATUS[429].EXT.BIT19 := FALSE;
   STATUS[429].EXT.BIT20 := FALSE;
   STATUS[429].EXT.AlarmSuppressed := FALSE;
   STATUS[429].EXT.AlarmPresent := FALSE;
   STATUS[429].EXT.AlarmFailUnAck := FALSE;
   STATUS[429].Status := 0;
   STATUS[429].TimeStamp := 16#0000;
   STATUS[430].EXT.AlarmWarnUnAck := FALSE;
   STATUS[430].EXT.AckRequired := FALSE;
   STATUS[430].EXT.Maintanence := FALSE;
   STATUS[430].EXT.Operation := FALSE;
   STATUS[430].EXT.Forced := FALSE;
   STATUS[430].EXT.BIT29 := FALSE;
   STATUS[430].EXT.BIT30 := FALSE;
   STATUS[430].EXT.BIT31 := FALSE;
   STATUS[430].EXT.ModeBit1 := FALSE;
   STATUS[430].EXT.ModeBit2 := FALSE;
   STATUS[430].EXT.ModeBit3 := FALSE;
   STATUS[430].EXT.BIT19 := FALSE;
   STATUS[430].EXT.BIT20 := FALSE;
   STATUS[430].EXT.AlarmSuppressed := FALSE;
   STATUS[430].EXT.AlarmPresent := FALSE;
   STATUS[430].EXT.AlarmFailUnAck := FALSE;
   STATUS[430].Status := 0;
   STATUS[430].TimeStamp := 16#0000;
   STATUS[431].EXT.AlarmWarnUnAck := FALSE;
   STATUS[431].EXT.AckRequired := FALSE;
   STATUS[431].EXT.Maintanence := FALSE;
   STATUS[431].EXT.Operation := FALSE;
   STATUS[431].EXT.Forced := FALSE;
   STATUS[431].EXT.BIT29 := FALSE;
   STATUS[431].EXT.BIT30 := FALSE;
   STATUS[431].EXT.BIT31 := FALSE;
   STATUS[431].EXT.ModeBit1 := FALSE;
   STATUS[431].EXT.ModeBit2 := FALSE;
   STATUS[431].EXT.ModeBit3 := FALSE;
   STATUS[431].EXT.BIT19 := FALSE;
   STATUS[431].EXT.BIT20 := FALSE;
   STATUS[431].EXT.AlarmSuppressed := FALSE;
   STATUS[431].EXT.AlarmPresent := FALSE;
   STATUS[431].EXT.AlarmFailUnAck := FALSE;
   STATUS[431].Status := 0;
   STATUS[431].TimeStamp := 16#0000;
   STATUS[432].EXT.AlarmWarnUnAck := FALSE;
   STATUS[432].EXT.AckRequired := FALSE;
   STATUS[432].EXT.Maintanence := FALSE;
   STATUS[432].EXT.Operation := FALSE;
   STATUS[432].EXT.Forced := FALSE;
   STATUS[432].EXT.BIT29 := FALSE;
   STATUS[432].EXT.BIT30 := FALSE;
   STATUS[432].EXT.BIT31 := FALSE;
   STATUS[432].EXT.ModeBit1 := FALSE;
   STATUS[432].EXT.ModeBit2 := FALSE;
   STATUS[432].EXT.ModeBit3 := FALSE;
   STATUS[432].EXT.BIT19 := FALSE;
   STATUS[432].EXT.BIT20 := FALSE;
   STATUS[432].EXT.AlarmSuppressed := FALSE;
   STATUS[432].EXT.AlarmPresent := FALSE;
   STATUS[432].EXT.AlarmFailUnAck := FALSE;
   STATUS[432].Status := 0;
   STATUS[432].TimeStamp := 16#0000;
   STATUS[433].EXT.AlarmWarnUnAck := FALSE;
   STATUS[433].EXT.AckRequired := FALSE;
   STATUS[433].EXT.Maintanence := FALSE;
   STATUS[433].EXT.Operation := FALSE;
   STATUS[433].EXT.Forced := FALSE;
   STATUS[433].EXT.BIT29 := FALSE;
   STATUS[433].EXT.BIT30 := FALSE;
   STATUS[433].EXT.BIT31 := FALSE;
   STATUS[433].EXT.ModeBit1 := FALSE;
   STATUS[433].EXT.ModeBit2 := FALSE;
   STATUS[433].EXT.ModeBit3 := FALSE;
   STATUS[433].EXT.BIT19 := FALSE;
   STATUS[433].EXT.BIT20 := FALSE;
   STATUS[433].EXT.AlarmSuppressed := FALSE;
   STATUS[433].EXT.AlarmPresent := FALSE;
   STATUS[433].EXT.AlarmFailUnAck := FALSE;
   STATUS[433].Status := 0;
   STATUS[433].TimeStamp := 16#0000;
   STATUS[434].EXT.AlarmWarnUnAck := FALSE;
   STATUS[434].EXT.AckRequired := FALSE;
   STATUS[434].EXT.Maintanence := FALSE;
   STATUS[434].EXT.Operation := FALSE;
   STATUS[434].EXT.Forced := FALSE;
   STATUS[434].EXT.BIT29 := FALSE;
   STATUS[434].EXT.BIT30 := FALSE;
   STATUS[434].EXT.BIT31 := FALSE;
   STATUS[434].EXT.ModeBit1 := TRUE;
   STATUS[434].EXT.ModeBit2 := TRUE;
   STATUS[434].EXT.ModeBit3 := FALSE;
   STATUS[434].EXT.BIT19 := FALSE;
   STATUS[434].EXT.BIT20 := FALSE;
   STATUS[434].EXT.AlarmSuppressed := FALSE;
   STATUS[434].EXT.AlarmPresent := TRUE;
   STATUS[434].EXT.AlarmFailUnAck := TRUE;
   STATUS[434].Status := 210;
   STATUS[434].TimeStamp := 16#1B30;
   STATUS[435].EXT.AlarmWarnUnAck := FALSE;
   STATUS[435].EXT.AckRequired := FALSE;
   STATUS[435].EXT.Maintanence := FALSE;
   STATUS[435].EXT.Operation := FALSE;
   STATUS[435].EXT.Forced := FALSE;
   STATUS[435].EXT.BIT29 := FALSE;
   STATUS[435].EXT.BIT30 := FALSE;
   STATUS[435].EXT.BIT31 := FALSE;
   STATUS[435].EXT.ModeBit1 := FALSE;
   STATUS[435].EXT.ModeBit2 := FALSE;
   STATUS[435].EXT.ModeBit3 := FALSE;
   STATUS[435].EXT.BIT19 := FALSE;
   STATUS[435].EXT.BIT20 := FALSE;
   STATUS[435].EXT.AlarmSuppressed := FALSE;
   STATUS[435].EXT.AlarmPresent := FALSE;
   STATUS[435].EXT.AlarmFailUnAck := FALSE;
   STATUS[435].Status := 0;
   STATUS[435].TimeStamp := 16#0000;
   STATUS[436].EXT.AlarmWarnUnAck := FALSE;
   STATUS[436].EXT.AckRequired := FALSE;
   STATUS[436].EXT.Maintanence := FALSE;
   STATUS[436].EXT.Operation := FALSE;
   STATUS[436].EXT.Forced := FALSE;
   STATUS[436].EXT.BIT29 := FALSE;
   STATUS[436].EXT.BIT30 := FALSE;
   STATUS[436].EXT.BIT31 := FALSE;
   STATUS[436].EXT.ModeBit1 := FALSE;
   STATUS[436].EXT.ModeBit2 := FALSE;
   STATUS[436].EXT.ModeBit3 := FALSE;
   STATUS[436].EXT.BIT19 := FALSE;
   STATUS[436].EXT.BIT20 := FALSE;
   STATUS[436].EXT.AlarmSuppressed := FALSE;
   STATUS[436].EXT.AlarmPresent := FALSE;
   STATUS[436].EXT.AlarmFailUnAck := FALSE;
   STATUS[436].Status := 0;
   STATUS[436].TimeStamp := 16#0000;
   STATUS[437].EXT.AlarmWarnUnAck := FALSE;
   STATUS[437].EXT.AckRequired := FALSE;
   STATUS[437].EXT.Maintanence := FALSE;
   STATUS[437].EXT.Operation := FALSE;
   STATUS[437].EXT.Forced := FALSE;
   STATUS[437].EXT.BIT29 := FALSE;
   STATUS[437].EXT.BIT30 := FALSE;
   STATUS[437].EXT.BIT31 := FALSE;
   STATUS[437].EXT.ModeBit1 := FALSE;
   STATUS[437].EXT.ModeBit2 := FALSE;
   STATUS[437].EXT.ModeBit3 := FALSE;
   STATUS[437].EXT.BIT19 := FALSE;
   STATUS[437].EXT.BIT20 := FALSE;
   STATUS[437].EXT.AlarmSuppressed := FALSE;
   STATUS[437].EXT.AlarmPresent := FALSE;
   STATUS[437].EXT.AlarmFailUnAck := FALSE;
   STATUS[437].Status := 0;
   STATUS[437].TimeStamp := 16#0000;
   STATUS[438].EXT.AlarmWarnUnAck := FALSE;
   STATUS[438].EXT.AckRequired := FALSE;
   STATUS[438].EXT.Maintanence := FALSE;
   STATUS[438].EXT.Operation := FALSE;
   STATUS[438].EXT.Forced := FALSE;
   STATUS[438].EXT.BIT29 := FALSE;
   STATUS[438].EXT.BIT30 := FALSE;
   STATUS[438].EXT.BIT31 := FALSE;
   STATUS[438].EXT.ModeBit1 := FALSE;
   STATUS[438].EXT.ModeBit2 := FALSE;
   STATUS[438].EXT.ModeBit3 := FALSE;
   STATUS[438].EXT.BIT19 := FALSE;
   STATUS[438].EXT.BIT20 := FALSE;
   STATUS[438].EXT.AlarmSuppressed := FALSE;
   STATUS[438].EXT.AlarmPresent := FALSE;
   STATUS[438].EXT.AlarmFailUnAck := FALSE;
   STATUS[438].Status := 0;
   STATUS[438].TimeStamp := 16#0000;
   STATUS[439].EXT.AlarmWarnUnAck := FALSE;
   STATUS[439].EXT.AckRequired := FALSE;
   STATUS[439].EXT.Maintanence := FALSE;
   STATUS[439].EXT.Operation := FALSE;
   STATUS[439].EXT.Forced := FALSE;
   STATUS[439].EXT.BIT29 := FALSE;
   STATUS[439].EXT.BIT30 := FALSE;
   STATUS[439].EXT.BIT31 := FALSE;
   STATUS[439].EXT.ModeBit1 := FALSE;
   STATUS[439].EXT.ModeBit2 := FALSE;
   STATUS[439].EXT.ModeBit3 := FALSE;
   STATUS[439].EXT.BIT19 := FALSE;
   STATUS[439].EXT.BIT20 := FALSE;
   STATUS[439].EXT.AlarmSuppressed := FALSE;
   STATUS[439].EXT.AlarmPresent := FALSE;
   STATUS[439].EXT.AlarmFailUnAck := FALSE;
   STATUS[439].Status := 0;
   STATUS[439].TimeStamp := 16#0000;
   STATUS[440].EXT.AlarmWarnUnAck := FALSE;
   STATUS[440].EXT.AckRequired := FALSE;
   STATUS[440].EXT.Maintanence := FALSE;
   STATUS[440].EXT.Operation := FALSE;
   STATUS[440].EXT.Forced := FALSE;
   STATUS[440].EXT.BIT29 := FALSE;
   STATUS[440].EXT.BIT30 := FALSE;
   STATUS[440].EXT.BIT31 := FALSE;
   STATUS[440].EXT.ModeBit1 := FALSE;
   STATUS[440].EXT.ModeBit2 := FALSE;
   STATUS[440].EXT.ModeBit3 := FALSE;
   STATUS[440].EXT.BIT19 := FALSE;
   STATUS[440].EXT.BIT20 := FALSE;
   STATUS[440].EXT.AlarmSuppressed := FALSE;
   STATUS[440].EXT.AlarmPresent := FALSE;
   STATUS[440].EXT.AlarmFailUnAck := FALSE;
   STATUS[440].Status := 0;
   STATUS[440].TimeStamp := 16#0000;
   STATUS[441].EXT.AlarmWarnUnAck := FALSE;
   STATUS[441].EXT.AckRequired := FALSE;
   STATUS[441].EXT.Maintanence := FALSE;
   STATUS[441].EXT.Operation := FALSE;
   STATUS[441].EXT.Forced := FALSE;
   STATUS[441].EXT.BIT29 := FALSE;
   STATUS[441].EXT.BIT30 := FALSE;
   STATUS[441].EXT.BIT31 := FALSE;
   STATUS[441].EXT.ModeBit1 := FALSE;
   STATUS[441].EXT.ModeBit2 := FALSE;
   STATUS[441].EXT.ModeBit3 := FALSE;
   STATUS[441].EXT.BIT19 := FALSE;
   STATUS[441].EXT.BIT20 := FALSE;
   STATUS[441].EXT.AlarmSuppressed := FALSE;
   STATUS[441].EXT.AlarmPresent := FALSE;
   STATUS[441].EXT.AlarmFailUnAck := FALSE;
   STATUS[441].Status := 0;
   STATUS[441].TimeStamp := 16#0000;
   STATUS[442].EXT.AlarmWarnUnAck := FALSE;
   STATUS[442].EXT.AckRequired := FALSE;
   STATUS[442].EXT.Maintanence := FALSE;
   STATUS[442].EXT.Operation := FALSE;
   STATUS[442].EXT.Forced := FALSE;
   STATUS[442].EXT.BIT29 := FALSE;
   STATUS[442].EXT.BIT30 := FALSE;
   STATUS[442].EXT.BIT31 := FALSE;
   STATUS[442].EXT.ModeBit1 := FALSE;
   STATUS[442].EXT.ModeBit2 := FALSE;
   STATUS[442].EXT.ModeBit3 := FALSE;
   STATUS[442].EXT.BIT19 := FALSE;
   STATUS[442].EXT.BIT20 := FALSE;
   STATUS[442].EXT.AlarmSuppressed := FALSE;
   STATUS[442].EXT.AlarmPresent := FALSE;
   STATUS[442].EXT.AlarmFailUnAck := FALSE;
   STATUS[442].Status := 0;
   STATUS[442].TimeStamp := 16#0000;
   STATUS[443].EXT.AlarmWarnUnAck := FALSE;
   STATUS[443].EXT.AckRequired := FALSE;
   STATUS[443].EXT.Maintanence := FALSE;
   STATUS[443].EXT.Operation := FALSE;
   STATUS[443].EXT.Forced := FALSE;
   STATUS[443].EXT.BIT29 := FALSE;
   STATUS[443].EXT.BIT30 := FALSE;
   STATUS[443].EXT.BIT31 := FALSE;
   STATUS[443].EXT.ModeBit1 := FALSE;
   STATUS[443].EXT.ModeBit2 := FALSE;
   STATUS[443].EXT.ModeBit3 := FALSE;
   STATUS[443].EXT.BIT19 := FALSE;
   STATUS[443].EXT.BIT20 := FALSE;
   STATUS[443].EXT.AlarmSuppressed := FALSE;
   STATUS[443].EXT.AlarmPresent := FALSE;
   STATUS[443].EXT.AlarmFailUnAck := FALSE;
   STATUS[443].Status := 0;
   STATUS[443].TimeStamp := 16#0000;
   STATUS[444].EXT.AlarmWarnUnAck := FALSE;
   STATUS[444].EXT.AckRequired := FALSE;
   STATUS[444].EXT.Maintanence := FALSE;
   STATUS[444].EXT.Operation := FALSE;
   STATUS[444].EXT.Forced := FALSE;
   STATUS[444].EXT.BIT29 := FALSE;
   STATUS[444].EXT.BIT30 := FALSE;
   STATUS[444].EXT.BIT31 := FALSE;
   STATUS[444].EXT.ModeBit1 := FALSE;
   STATUS[444].EXT.ModeBit2 := FALSE;
   STATUS[444].EXT.ModeBit3 := FALSE;
   STATUS[444].EXT.BIT19 := FALSE;
   STATUS[444].EXT.BIT20 := FALSE;
   STATUS[444].EXT.AlarmSuppressed := FALSE;
   STATUS[444].EXT.AlarmPresent := FALSE;
   STATUS[444].EXT.AlarmFailUnAck := FALSE;
   STATUS[444].Status := 0;
   STATUS[444].TimeStamp := 16#0000;
   STATUS[445].EXT.AlarmWarnUnAck := FALSE;
   STATUS[445].EXT.AckRequired := FALSE;
   STATUS[445].EXT.Maintanence := FALSE;
   STATUS[445].EXT.Operation := FALSE;
   STATUS[445].EXT.Forced := FALSE;
   STATUS[445].EXT.BIT29 := FALSE;
   STATUS[445].EXT.BIT30 := FALSE;
   STATUS[445].EXT.BIT31 := FALSE;
   STATUS[445].EXT.ModeBit1 := FALSE;
   STATUS[445].EXT.ModeBit2 := FALSE;
   STATUS[445].EXT.ModeBit3 := FALSE;
   STATUS[445].EXT.BIT19 := FALSE;
   STATUS[445].EXT.BIT20 := FALSE;
   STATUS[445].EXT.AlarmSuppressed := FALSE;
   STATUS[445].EXT.AlarmPresent := FALSE;
   STATUS[445].EXT.AlarmFailUnAck := FALSE;
   STATUS[445].Status := 0;
   STATUS[445].TimeStamp := 16#0000;
   STATUS[446].EXT.AlarmWarnUnAck := FALSE;
   STATUS[446].EXT.AckRequired := FALSE;
   STATUS[446].EXT.Maintanence := FALSE;
   STATUS[446].EXT.Operation := FALSE;
   STATUS[446].EXT.Forced := FALSE;
   STATUS[446].EXT.BIT29 := FALSE;
   STATUS[446].EXT.BIT30 := FALSE;
   STATUS[446].EXT.BIT31 := FALSE;
   STATUS[446].EXT.ModeBit1 := FALSE;
   STATUS[446].EXT.ModeBit2 := FALSE;
   STATUS[446].EXT.ModeBit3 := FALSE;
   STATUS[446].EXT.BIT19 := FALSE;
   STATUS[446].EXT.BIT20 := FALSE;
   STATUS[446].EXT.AlarmSuppressed := FALSE;
   STATUS[446].EXT.AlarmPresent := FALSE;
   STATUS[446].EXT.AlarmFailUnAck := FALSE;
   STATUS[446].Status := 0;
   STATUS[446].TimeStamp := 16#0000;
   STATUS[447].EXT.AlarmWarnUnAck := FALSE;
   STATUS[447].EXT.AckRequired := FALSE;
   STATUS[447].EXT.Maintanence := FALSE;
   STATUS[447].EXT.Operation := FALSE;
   STATUS[447].EXT.Forced := FALSE;
   STATUS[447].EXT.BIT29 := FALSE;
   STATUS[447].EXT.BIT30 := FALSE;
   STATUS[447].EXT.BIT31 := FALSE;
   STATUS[447].EXT.ModeBit1 := FALSE;
   STATUS[447].EXT.ModeBit2 := FALSE;
   STATUS[447].EXT.ModeBit3 := FALSE;
   STATUS[447].EXT.BIT19 := FALSE;
   STATUS[447].EXT.BIT20 := FALSE;
   STATUS[447].EXT.AlarmSuppressed := FALSE;
   STATUS[447].EXT.AlarmPresent := FALSE;
   STATUS[447].EXT.AlarmFailUnAck := FALSE;
   STATUS[447].Status := 0;
   STATUS[447].TimeStamp := 16#0000;
   STATUS[448].EXT.AlarmWarnUnAck := FALSE;
   STATUS[448].EXT.AckRequired := FALSE;
   STATUS[448].EXT.Maintanence := FALSE;
   STATUS[448].EXT.Operation := FALSE;
   STATUS[448].EXT.Forced := FALSE;
   STATUS[448].EXT.BIT29 := FALSE;
   STATUS[448].EXT.BIT30 := FALSE;
   STATUS[448].EXT.BIT31 := FALSE;
   STATUS[448].EXT.ModeBit1 := FALSE;
   STATUS[448].EXT.ModeBit2 := FALSE;
   STATUS[448].EXT.ModeBit3 := FALSE;
   STATUS[448].EXT.BIT19 := FALSE;
   STATUS[448].EXT.BIT20 := FALSE;
   STATUS[448].EXT.AlarmSuppressed := FALSE;
   STATUS[448].EXT.AlarmPresent := FALSE;
   STATUS[448].EXT.AlarmFailUnAck := FALSE;
   STATUS[448].Status := 0;
   STATUS[448].TimeStamp := 16#0000;
   STATUS[449].EXT.AlarmWarnUnAck := FALSE;
   STATUS[449].EXT.AckRequired := FALSE;
   STATUS[449].EXT.Maintanence := FALSE;
   STATUS[449].EXT.Operation := FALSE;
   STATUS[449].EXT.Forced := FALSE;
   STATUS[449].EXT.BIT29 := FALSE;
   STATUS[449].EXT.BIT30 := FALSE;
   STATUS[449].EXT.BIT31 := FALSE;
   STATUS[449].EXT.ModeBit1 := FALSE;
   STATUS[449].EXT.ModeBit2 := FALSE;
   STATUS[449].EXT.ModeBit3 := FALSE;
   STATUS[449].EXT.BIT19 := FALSE;
   STATUS[449].EXT.BIT20 := FALSE;
   STATUS[449].EXT.AlarmSuppressed := FALSE;
   STATUS[449].EXT.AlarmPresent := FALSE;
   STATUS[449].EXT.AlarmFailUnAck := FALSE;
   STATUS[449].Status := 0;
   STATUS[449].TimeStamp := 16#0000;
   STATUS[450].EXT.AlarmWarnUnAck := FALSE;
   STATUS[450].EXT.AckRequired := FALSE;
   STATUS[450].EXT.Maintanence := FALSE;
   STATUS[450].EXT.Operation := FALSE;
   STATUS[450].EXT.Forced := FALSE;
   STATUS[450].EXT.BIT29 := FALSE;
   STATUS[450].EXT.BIT30 := FALSE;
   STATUS[450].EXT.BIT31 := FALSE;
   STATUS[450].EXT.ModeBit1 := FALSE;
   STATUS[450].EXT.ModeBit2 := FALSE;
   STATUS[450].EXT.ModeBit3 := FALSE;
   STATUS[450].EXT.BIT19 := FALSE;
   STATUS[450].EXT.BIT20 := FALSE;
   STATUS[450].EXT.AlarmSuppressed := FALSE;
   STATUS[450].EXT.AlarmPresent := FALSE;
   STATUS[450].EXT.AlarmFailUnAck := FALSE;
   STATUS[450].Status := 0;
   STATUS[450].TimeStamp := 16#0000;
   STATUS[451].EXT.AlarmWarnUnAck := FALSE;
   STATUS[451].EXT.AckRequired := FALSE;
   STATUS[451].EXT.Maintanence := FALSE;
   STATUS[451].EXT.Operation := FALSE;
   STATUS[451].EXT.Forced := FALSE;
   STATUS[451].EXT.BIT29 := FALSE;
   STATUS[451].EXT.BIT30 := FALSE;
   STATUS[451].EXT.BIT31 := FALSE;
   STATUS[451].EXT.ModeBit1 := FALSE;
   STATUS[451].EXT.ModeBit2 := FALSE;
   STATUS[451].EXT.ModeBit3 := FALSE;
   STATUS[451].EXT.BIT19 := FALSE;
   STATUS[451].EXT.BIT20 := FALSE;
   STATUS[451].EXT.AlarmSuppressed := FALSE;
   STATUS[451].EXT.AlarmPresent := FALSE;
   STATUS[451].EXT.AlarmFailUnAck := FALSE;
   STATUS[451].Status := 0;
   STATUS[451].TimeStamp := 16#0000;
   STATUS[452].EXT.AlarmWarnUnAck := FALSE;
   STATUS[452].EXT.AckRequired := FALSE;
   STATUS[452].EXT.Maintanence := FALSE;
   STATUS[452].EXT.Operation := FALSE;
   STATUS[452].EXT.Forced := FALSE;
   STATUS[452].EXT.BIT29 := FALSE;
   STATUS[452].EXT.BIT30 := FALSE;
   STATUS[452].EXT.BIT31 := FALSE;
   STATUS[452].EXT.ModeBit1 := FALSE;
   STATUS[452].EXT.ModeBit2 := FALSE;
   STATUS[452].EXT.ModeBit3 := FALSE;
   STATUS[452].EXT.BIT19 := FALSE;
   STATUS[452].EXT.BIT20 := FALSE;
   STATUS[452].EXT.AlarmSuppressed := FALSE;
   STATUS[452].EXT.AlarmPresent := FALSE;
   STATUS[452].EXT.AlarmFailUnAck := FALSE;
   STATUS[452].Status := 0;
   STATUS[452].TimeStamp := 16#0000;
   STATUS[453].EXT.AlarmWarnUnAck := FALSE;
   STATUS[453].EXT.AckRequired := FALSE;
   STATUS[453].EXT.Maintanence := FALSE;
   STATUS[453].EXT.Operation := FALSE;
   STATUS[453].EXT.Forced := FALSE;
   STATUS[453].EXT.BIT29 := FALSE;
   STATUS[453].EXT.BIT30 := FALSE;
   STATUS[453].EXT.BIT31 := FALSE;
   STATUS[453].EXT.ModeBit1 := FALSE;
   STATUS[453].EXT.ModeBit2 := FALSE;
   STATUS[453].EXT.ModeBit3 := FALSE;
   STATUS[453].EXT.BIT19 := FALSE;
   STATUS[453].EXT.BIT20 := FALSE;
   STATUS[453].EXT.AlarmSuppressed := FALSE;
   STATUS[453].EXT.AlarmPresent := FALSE;
   STATUS[453].EXT.AlarmFailUnAck := FALSE;
   STATUS[453].Status := 0;
   STATUS[453].TimeStamp := 16#0000;
   STATUS[454].EXT.AlarmWarnUnAck := FALSE;
   STATUS[454].EXT.AckRequired := FALSE;
   STATUS[454].EXT.Maintanence := FALSE;
   STATUS[454].EXT.Operation := FALSE;
   STATUS[454].EXT.Forced := FALSE;
   STATUS[454].EXT.BIT29 := FALSE;
   STATUS[454].EXT.BIT30 := FALSE;
   STATUS[454].EXT.BIT31 := FALSE;
   STATUS[454].EXT.ModeBit1 := FALSE;
   STATUS[454].EXT.ModeBit2 := FALSE;
   STATUS[454].EXT.ModeBit3 := FALSE;
   STATUS[454].EXT.BIT19 := FALSE;
   STATUS[454].EXT.BIT20 := FALSE;
   STATUS[454].EXT.AlarmSuppressed := FALSE;
   STATUS[454].EXT.AlarmPresent := FALSE;
   STATUS[454].EXT.AlarmFailUnAck := FALSE;
   STATUS[454].Status := 0;
   STATUS[454].TimeStamp := 16#0000;
   STATUS[455].EXT.AlarmWarnUnAck := FALSE;
   STATUS[455].EXT.AckRequired := FALSE;
   STATUS[455].EXT.Maintanence := FALSE;
   STATUS[455].EXT.Operation := FALSE;
   STATUS[455].EXT.Forced := FALSE;
   STATUS[455].EXT.BIT29 := FALSE;
   STATUS[455].EXT.BIT30 := FALSE;
   STATUS[455].EXT.BIT31 := FALSE;
   STATUS[455].EXT.ModeBit1 := FALSE;
   STATUS[455].EXT.ModeBit2 := FALSE;
   STATUS[455].EXT.ModeBit3 := FALSE;
   STATUS[455].EXT.BIT19 := FALSE;
   STATUS[455].EXT.BIT20 := FALSE;
   STATUS[455].EXT.AlarmSuppressed := FALSE;
   STATUS[455].EXT.AlarmPresent := FALSE;
   STATUS[455].EXT.AlarmFailUnAck := FALSE;
   STATUS[455].Status := 0;
   STATUS[455].TimeStamp := 16#0000;
   STATUS[456].EXT.AlarmWarnUnAck := FALSE;
   STATUS[456].EXT.AckRequired := FALSE;
   STATUS[456].EXT.Maintanence := FALSE;
   STATUS[456].EXT.Operation := FALSE;
   STATUS[456].EXT.Forced := FALSE;
   STATUS[456].EXT.BIT29 := FALSE;
   STATUS[456].EXT.BIT30 := FALSE;
   STATUS[456].EXT.BIT31 := FALSE;
   STATUS[456].EXT.ModeBit1 := FALSE;
   STATUS[456].EXT.ModeBit2 := FALSE;
   STATUS[456].EXT.ModeBit3 := FALSE;
   STATUS[456].EXT.BIT19 := FALSE;
   STATUS[456].EXT.BIT20 := FALSE;
   STATUS[456].EXT.AlarmSuppressed := FALSE;
   STATUS[456].EXT.AlarmPresent := FALSE;
   STATUS[456].EXT.AlarmFailUnAck := FALSE;
   STATUS[456].Status := 0;
   STATUS[456].TimeStamp := 16#0000;
   STATUS[457].EXT.AlarmWarnUnAck := FALSE;
   STATUS[457].EXT.AckRequired := FALSE;
   STATUS[457].EXT.Maintanence := FALSE;
   STATUS[457].EXT.Operation := FALSE;
   STATUS[457].EXT.Forced := FALSE;
   STATUS[457].EXT.BIT29 := FALSE;
   STATUS[457].EXT.BIT30 := FALSE;
   STATUS[457].EXT.BIT31 := FALSE;
   STATUS[457].EXT.ModeBit1 := FALSE;
   STATUS[457].EXT.ModeBit2 := FALSE;
   STATUS[457].EXT.ModeBit3 := FALSE;
   STATUS[457].EXT.BIT19 := FALSE;
   STATUS[457].EXT.BIT20 := FALSE;
   STATUS[457].EXT.AlarmSuppressed := FALSE;
   STATUS[457].EXT.AlarmPresent := FALSE;
   STATUS[457].EXT.AlarmFailUnAck := FALSE;
   STATUS[457].Status := 0;
   STATUS[457].TimeStamp := 16#0000;
   STATUS[458].EXT.AlarmWarnUnAck := FALSE;
   STATUS[458].EXT.AckRequired := FALSE;
   STATUS[458].EXT.Maintanence := FALSE;
   STATUS[458].EXT.Operation := FALSE;
   STATUS[458].EXT.Forced := FALSE;
   STATUS[458].EXT.BIT29 := FALSE;
   STATUS[458].EXT.BIT30 := FALSE;
   STATUS[458].EXT.BIT31 := FALSE;
   STATUS[458].EXT.ModeBit1 := FALSE;
   STATUS[458].EXT.ModeBit2 := FALSE;
   STATUS[458].EXT.ModeBit3 := FALSE;
   STATUS[458].EXT.BIT19 := FALSE;
   STATUS[458].EXT.BIT20 := FALSE;
   STATUS[458].EXT.AlarmSuppressed := FALSE;
   STATUS[458].EXT.AlarmPresent := FALSE;
   STATUS[458].EXT.AlarmFailUnAck := FALSE;
   STATUS[458].Status := 0;
   STATUS[458].TimeStamp := 16#0000;
   STATUS[459].EXT.AlarmWarnUnAck := FALSE;
   STATUS[459].EXT.AckRequired := FALSE;
   STATUS[459].EXT.Maintanence := FALSE;
   STATUS[459].EXT.Operation := FALSE;
   STATUS[459].EXT.Forced := FALSE;
   STATUS[459].EXT.BIT29 := FALSE;
   STATUS[459].EXT.BIT30 := FALSE;
   STATUS[459].EXT.BIT31 := FALSE;
   STATUS[459].EXT.ModeBit1 := FALSE;
   STATUS[459].EXT.ModeBit2 := FALSE;
   STATUS[459].EXT.ModeBit3 := FALSE;
   STATUS[459].EXT.BIT19 := FALSE;
   STATUS[459].EXT.BIT20 := FALSE;
   STATUS[459].EXT.AlarmSuppressed := FALSE;
   STATUS[459].EXT.AlarmPresent := FALSE;
   STATUS[459].EXT.AlarmFailUnAck := FALSE;
   STATUS[459].Status := 0;
   STATUS[459].TimeStamp := 16#0000;
   STATUS[460].EXT.AlarmWarnUnAck := FALSE;
   STATUS[460].EXT.AckRequired := FALSE;
   STATUS[460].EXT.Maintanence := FALSE;
   STATUS[460].EXT.Operation := FALSE;
   STATUS[460].EXT.Forced := FALSE;
   STATUS[460].EXT.BIT29 := FALSE;
   STATUS[460].EXT.BIT30 := FALSE;
   STATUS[460].EXT.BIT31 := FALSE;
   STATUS[460].EXT.ModeBit1 := FALSE;
   STATUS[460].EXT.ModeBit2 := FALSE;
   STATUS[460].EXT.ModeBit3 := FALSE;
   STATUS[460].EXT.BIT19 := FALSE;
   STATUS[460].EXT.BIT20 := FALSE;
   STATUS[460].EXT.AlarmSuppressed := FALSE;
   STATUS[460].EXT.AlarmPresent := FALSE;
   STATUS[460].EXT.AlarmFailUnAck := FALSE;
   STATUS[460].Status := 0;
   STATUS[460].TimeStamp := 16#0000;
   STATUS[461].EXT.AlarmWarnUnAck := FALSE;
   STATUS[461].EXT.AckRequired := FALSE;
   STATUS[461].EXT.Maintanence := FALSE;
   STATUS[461].EXT.Operation := FALSE;
   STATUS[461].EXT.Forced := FALSE;
   STATUS[461].EXT.BIT29 := FALSE;
   STATUS[461].EXT.BIT30 := FALSE;
   STATUS[461].EXT.BIT31 := FALSE;
   STATUS[461].EXT.ModeBit1 := FALSE;
   STATUS[461].EXT.ModeBit2 := FALSE;
   STATUS[461].EXT.ModeBit3 := FALSE;
   STATUS[461].EXT.BIT19 := FALSE;
   STATUS[461].EXT.BIT20 := FALSE;
   STATUS[461].EXT.AlarmSuppressed := FALSE;
   STATUS[461].EXT.AlarmPresent := FALSE;
   STATUS[461].EXT.AlarmFailUnAck := FALSE;
   STATUS[461].Status := 0;
   STATUS[461].TimeStamp := 16#0000;
   STATUS[462].EXT.AlarmWarnUnAck := FALSE;
   STATUS[462].EXT.AckRequired := FALSE;
   STATUS[462].EXT.Maintanence := FALSE;
   STATUS[462].EXT.Operation := FALSE;
   STATUS[462].EXT.Forced := FALSE;
   STATUS[462].EXT.BIT29 := FALSE;
   STATUS[462].EXT.BIT30 := FALSE;
   STATUS[462].EXT.BIT31 := FALSE;
   STATUS[462].EXT.ModeBit1 := FALSE;
   STATUS[462].EXT.ModeBit2 := FALSE;
   STATUS[462].EXT.ModeBit3 := FALSE;
   STATUS[462].EXT.BIT19 := FALSE;
   STATUS[462].EXT.BIT20 := FALSE;
   STATUS[462].EXT.AlarmSuppressed := FALSE;
   STATUS[462].EXT.AlarmPresent := FALSE;
   STATUS[462].EXT.AlarmFailUnAck := FALSE;
   STATUS[462].Status := 0;
   STATUS[462].TimeStamp := 16#0000;
   STATUS[463].EXT.AlarmWarnUnAck := FALSE;
   STATUS[463].EXT.AckRequired := FALSE;
   STATUS[463].EXT.Maintanence := FALSE;
   STATUS[463].EXT.Operation := FALSE;
   STATUS[463].EXT.Forced := FALSE;
   STATUS[463].EXT.BIT29 := FALSE;
   STATUS[463].EXT.BIT30 := FALSE;
   STATUS[463].EXT.BIT31 := FALSE;
   STATUS[463].EXT.ModeBit1 := FALSE;
   STATUS[463].EXT.ModeBit2 := FALSE;
   STATUS[463].EXT.ModeBit3 := FALSE;
   STATUS[463].EXT.BIT19 := FALSE;
   STATUS[463].EXT.BIT20 := FALSE;
   STATUS[463].EXT.AlarmSuppressed := FALSE;
   STATUS[463].EXT.AlarmPresent := FALSE;
   STATUS[463].EXT.AlarmFailUnAck := FALSE;
   STATUS[463].Status := 0;
   STATUS[463].TimeStamp := 16#0000;
   STATUS[464].EXT.AlarmWarnUnAck := FALSE;
   STATUS[464].EXT.AckRequired := FALSE;
   STATUS[464].EXT.Maintanence := FALSE;
   STATUS[464].EXT.Operation := FALSE;
   STATUS[464].EXT.Forced := FALSE;
   STATUS[464].EXT.BIT29 := FALSE;
   STATUS[464].EXT.BIT30 := FALSE;
   STATUS[464].EXT.BIT31 := FALSE;
   STATUS[464].EXT.ModeBit1 := FALSE;
   STATUS[464].EXT.ModeBit2 := FALSE;
   STATUS[464].EXT.ModeBit3 := FALSE;
   STATUS[464].EXT.BIT19 := FALSE;
   STATUS[464].EXT.BIT20 := FALSE;
   STATUS[464].EXT.AlarmSuppressed := FALSE;
   STATUS[464].EXT.AlarmPresent := FALSE;
   STATUS[464].EXT.AlarmFailUnAck := FALSE;
   STATUS[464].Status := 0;
   STATUS[464].TimeStamp := 16#0000;
   STATUS[465].EXT.AlarmWarnUnAck := FALSE;
   STATUS[465].EXT.AckRequired := FALSE;
   STATUS[465].EXT.Maintanence := FALSE;
   STATUS[465].EXT.Operation := FALSE;
   STATUS[465].EXT.Forced := FALSE;
   STATUS[465].EXT.BIT29 := FALSE;
   STATUS[465].EXT.BIT30 := FALSE;
   STATUS[465].EXT.BIT31 := FALSE;
   STATUS[465].EXT.ModeBit1 := FALSE;
   STATUS[465].EXT.ModeBit2 := FALSE;
   STATUS[465].EXT.ModeBit3 := FALSE;
   STATUS[465].EXT.BIT19 := FALSE;
   STATUS[465].EXT.BIT20 := FALSE;
   STATUS[465].EXT.AlarmSuppressed := FALSE;
   STATUS[465].EXT.AlarmPresent := FALSE;
   STATUS[465].EXT.AlarmFailUnAck := FALSE;
   STATUS[465].Status := 0;
   STATUS[465].TimeStamp := 16#0000;
   STATUS[466].EXT.AlarmWarnUnAck := FALSE;
   STATUS[466].EXT.AckRequired := FALSE;
   STATUS[466].EXT.Maintanence := FALSE;
   STATUS[466].EXT.Operation := FALSE;
   STATUS[466].EXT.Forced := FALSE;
   STATUS[466].EXT.BIT29 := FALSE;
   STATUS[466].EXT.BIT30 := FALSE;
   STATUS[466].EXT.BIT31 := FALSE;
   STATUS[466].EXT.ModeBit1 := FALSE;
   STATUS[466].EXT.ModeBit2 := FALSE;
   STATUS[466].EXT.ModeBit3 := FALSE;
   STATUS[466].EXT.BIT19 := FALSE;
   STATUS[466].EXT.BIT20 := FALSE;
   STATUS[466].EXT.AlarmSuppressed := FALSE;
   STATUS[466].EXT.AlarmPresent := FALSE;
   STATUS[466].EXT.AlarmFailUnAck := FALSE;
   STATUS[466].Status := 0;
   STATUS[466].TimeStamp := 16#0000;
   STATUS[467].EXT.AlarmWarnUnAck := FALSE;
   STATUS[467].EXT.AckRequired := FALSE;
   STATUS[467].EXT.Maintanence := FALSE;
   STATUS[467].EXT.Operation := FALSE;
   STATUS[467].EXT.Forced := FALSE;
   STATUS[467].EXT.BIT29 := FALSE;
   STATUS[467].EXT.BIT30 := FALSE;
   STATUS[467].EXT.BIT31 := FALSE;
   STATUS[467].EXT.ModeBit1 := FALSE;
   STATUS[467].EXT.ModeBit2 := FALSE;
   STATUS[467].EXT.ModeBit3 := FALSE;
   STATUS[467].EXT.BIT19 := FALSE;
   STATUS[467].EXT.BIT20 := FALSE;
   STATUS[467].EXT.AlarmSuppressed := FALSE;
   STATUS[467].EXT.AlarmPresent := FALSE;
   STATUS[467].EXT.AlarmFailUnAck := FALSE;
   STATUS[467].Status := 0;
   STATUS[467].TimeStamp := 16#0000;
   STATUS[468].EXT.AlarmWarnUnAck := FALSE;
   STATUS[468].EXT.AckRequired := FALSE;
   STATUS[468].EXT.Maintanence := FALSE;
   STATUS[468].EXT.Operation := FALSE;
   STATUS[468].EXT.Forced := FALSE;
   STATUS[468].EXT.BIT29 := FALSE;
   STATUS[468].EXT.BIT30 := FALSE;
   STATUS[468].EXT.BIT31 := FALSE;
   STATUS[468].EXT.ModeBit1 := FALSE;
   STATUS[468].EXT.ModeBit2 := FALSE;
   STATUS[468].EXT.ModeBit3 := FALSE;
   STATUS[468].EXT.BIT19 := FALSE;
   STATUS[468].EXT.BIT20 := FALSE;
   STATUS[468].EXT.AlarmSuppressed := FALSE;
   STATUS[468].EXT.AlarmPresent := FALSE;
   STATUS[468].EXT.AlarmFailUnAck := FALSE;
   STATUS[468].Status := 0;
   STATUS[468].TimeStamp := 16#0000;
   STATUS[469].EXT.AlarmWarnUnAck := FALSE;
   STATUS[469].EXT.AckRequired := FALSE;
   STATUS[469].EXT.Maintanence := FALSE;
   STATUS[469].EXT.Operation := FALSE;
   STATUS[469].EXT.Forced := FALSE;
   STATUS[469].EXT.BIT29 := FALSE;
   STATUS[469].EXT.BIT30 := FALSE;
   STATUS[469].EXT.BIT31 := FALSE;
   STATUS[469].EXT.ModeBit1 := FALSE;
   STATUS[469].EXT.ModeBit2 := FALSE;
   STATUS[469].EXT.ModeBit3 := FALSE;
   STATUS[469].EXT.BIT19 := FALSE;
   STATUS[469].EXT.BIT20 := FALSE;
   STATUS[469].EXT.AlarmSuppressed := FALSE;
   STATUS[469].EXT.AlarmPresent := FALSE;
   STATUS[469].EXT.AlarmFailUnAck := FALSE;
   STATUS[469].Status := 0;
   STATUS[469].TimeStamp := 16#0000;
   STATUS[470].EXT.AlarmWarnUnAck := FALSE;
   STATUS[470].EXT.AckRequired := FALSE;
   STATUS[470].EXT.Maintanence := FALSE;
   STATUS[470].EXT.Operation := FALSE;
   STATUS[470].EXT.Forced := FALSE;
   STATUS[470].EXT.BIT29 := FALSE;
   STATUS[470].EXT.BIT30 := FALSE;
   STATUS[470].EXT.BIT31 := FALSE;
   STATUS[470].EXT.ModeBit1 := FALSE;
   STATUS[470].EXT.ModeBit2 := FALSE;
   STATUS[470].EXT.ModeBit3 := FALSE;
   STATUS[470].EXT.BIT19 := FALSE;
   STATUS[470].EXT.BIT20 := FALSE;
   STATUS[470].EXT.AlarmSuppressed := FALSE;
   STATUS[470].EXT.AlarmPresent := FALSE;
   STATUS[470].EXT.AlarmFailUnAck := FALSE;
   STATUS[470].Status := 0;
   STATUS[470].TimeStamp := 16#0000;
   STATUS[471].EXT.AlarmWarnUnAck := FALSE;
   STATUS[471].EXT.AckRequired := FALSE;
   STATUS[471].EXT.Maintanence := FALSE;
   STATUS[471].EXT.Operation := FALSE;
   STATUS[471].EXT.Forced := FALSE;
   STATUS[471].EXT.BIT29 := FALSE;
   STATUS[471].EXT.BIT30 := FALSE;
   STATUS[471].EXT.BIT31 := FALSE;
   STATUS[471].EXT.ModeBit1 := FALSE;
   STATUS[471].EXT.ModeBit2 := FALSE;
   STATUS[471].EXT.ModeBit3 := FALSE;
   STATUS[471].EXT.BIT19 := FALSE;
   STATUS[471].EXT.BIT20 := FALSE;
   STATUS[471].EXT.AlarmSuppressed := FALSE;
   STATUS[471].EXT.AlarmPresent := FALSE;
   STATUS[471].EXT.AlarmFailUnAck := FALSE;
   STATUS[471].Status := 0;
   STATUS[471].TimeStamp := 16#0000;
   STATUS[472].EXT.AlarmWarnUnAck := FALSE;
   STATUS[472].EXT.AckRequired := FALSE;
   STATUS[472].EXT.Maintanence := FALSE;
   STATUS[472].EXT.Operation := FALSE;
   STATUS[472].EXT.Forced := FALSE;
   STATUS[472].EXT.BIT29 := FALSE;
   STATUS[472].EXT.BIT30 := FALSE;
   STATUS[472].EXT.BIT31 := FALSE;
   STATUS[472].EXT.ModeBit1 := FALSE;
   STATUS[472].EXT.ModeBit2 := FALSE;
   STATUS[472].EXT.ModeBit3 := FALSE;
   STATUS[472].EXT.BIT19 := FALSE;
   STATUS[472].EXT.BIT20 := FALSE;
   STATUS[472].EXT.AlarmSuppressed := FALSE;
   STATUS[472].EXT.AlarmPresent := FALSE;
   STATUS[472].EXT.AlarmFailUnAck := FALSE;
   STATUS[472].Status := 0;
   STATUS[472].TimeStamp := 16#0000;
   STATUS[473].EXT.AlarmWarnUnAck := FALSE;
   STATUS[473].EXT.AckRequired := FALSE;
   STATUS[473].EXT.Maintanence := FALSE;
   STATUS[473].EXT.Operation := FALSE;
   STATUS[473].EXT.Forced := FALSE;
   STATUS[473].EXT.BIT29 := FALSE;
   STATUS[473].EXT.BIT30 := FALSE;
   STATUS[473].EXT.BIT31 := FALSE;
   STATUS[473].EXT.ModeBit1 := FALSE;
   STATUS[473].EXT.ModeBit2 := FALSE;
   STATUS[473].EXT.ModeBit3 := FALSE;
   STATUS[473].EXT.BIT19 := FALSE;
   STATUS[473].EXT.BIT20 := FALSE;
   STATUS[473].EXT.AlarmSuppressed := FALSE;
   STATUS[473].EXT.AlarmPresent := FALSE;
   STATUS[473].EXT.AlarmFailUnAck := FALSE;
   STATUS[473].Status := 0;
   STATUS[473].TimeStamp := 16#0000;
   STATUS[474].EXT.AlarmWarnUnAck := FALSE;
   STATUS[474].EXT.AckRequired := FALSE;
   STATUS[474].EXT.Maintanence := FALSE;
   STATUS[474].EXT.Operation := FALSE;
   STATUS[474].EXT.Forced := FALSE;
   STATUS[474].EXT.BIT29 := FALSE;
   STATUS[474].EXT.BIT30 := FALSE;
   STATUS[474].EXT.BIT31 := FALSE;
   STATUS[474].EXT.ModeBit1 := FALSE;
   STATUS[474].EXT.ModeBit2 := FALSE;
   STATUS[474].EXT.ModeBit3 := FALSE;
   STATUS[474].EXT.BIT19 := FALSE;
   STATUS[474].EXT.BIT20 := FALSE;
   STATUS[474].EXT.AlarmSuppressed := FALSE;
   STATUS[474].EXT.AlarmPresent := FALSE;
   STATUS[474].EXT.AlarmFailUnAck := FALSE;
   STATUS[474].Status := 0;
   STATUS[474].TimeStamp := 16#0000;
   STATUS[475].EXT.AlarmWarnUnAck := FALSE;
   STATUS[475].EXT.AckRequired := FALSE;
   STATUS[475].EXT.Maintanence := FALSE;
   STATUS[475].EXT.Operation := FALSE;
   STATUS[475].EXT.Forced := FALSE;
   STATUS[475].EXT.BIT29 := FALSE;
   STATUS[475].EXT.BIT30 := FALSE;
   STATUS[475].EXT.BIT31 := FALSE;
   STATUS[475].EXT.ModeBit1 := FALSE;
   STATUS[475].EXT.ModeBit2 := FALSE;
   STATUS[475].EXT.ModeBit3 := FALSE;
   STATUS[475].EXT.BIT19 := FALSE;
   STATUS[475].EXT.BIT20 := FALSE;
   STATUS[475].EXT.AlarmSuppressed := FALSE;
   STATUS[475].EXT.AlarmPresent := FALSE;
   STATUS[475].EXT.AlarmFailUnAck := FALSE;
   STATUS[475].Status := 0;
   STATUS[475].TimeStamp := 16#0000;
   STATUS[476].EXT.AlarmWarnUnAck := FALSE;
   STATUS[476].EXT.AckRequired := FALSE;
   STATUS[476].EXT.Maintanence := FALSE;
   STATUS[476].EXT.Operation := FALSE;
   STATUS[476].EXT.Forced := FALSE;
   STATUS[476].EXT.BIT29 := FALSE;
   STATUS[476].EXT.BIT30 := FALSE;
   STATUS[476].EXT.BIT31 := FALSE;
   STATUS[476].EXT.ModeBit1 := FALSE;
   STATUS[476].EXT.ModeBit2 := FALSE;
   STATUS[476].EXT.ModeBit3 := FALSE;
   STATUS[476].EXT.BIT19 := FALSE;
   STATUS[476].EXT.BIT20 := FALSE;
   STATUS[476].EXT.AlarmSuppressed := FALSE;
   STATUS[476].EXT.AlarmPresent := FALSE;
   STATUS[476].EXT.AlarmFailUnAck := FALSE;
   STATUS[476].Status := 0;
   STATUS[476].TimeStamp := 16#0000;
   STATUS[477].EXT.AlarmWarnUnAck := FALSE;
   STATUS[477].EXT.AckRequired := FALSE;
   STATUS[477].EXT.Maintanence := FALSE;
   STATUS[477].EXT.Operation := FALSE;
   STATUS[477].EXT.Forced := FALSE;
   STATUS[477].EXT.BIT29 := FALSE;
   STATUS[477].EXT.BIT30 := FALSE;
   STATUS[477].EXT.BIT31 := FALSE;
   STATUS[477].EXT.ModeBit1 := FALSE;
   STATUS[477].EXT.ModeBit2 := FALSE;
   STATUS[477].EXT.ModeBit3 := FALSE;
   STATUS[477].EXT.BIT19 := FALSE;
   STATUS[477].EXT.BIT20 := FALSE;
   STATUS[477].EXT.AlarmSuppressed := FALSE;
   STATUS[477].EXT.AlarmPresent := FALSE;
   STATUS[477].EXT.AlarmFailUnAck := FALSE;
   STATUS[477].Status := 0;
   STATUS[477].TimeStamp := 16#0000;
   STATUS[478].EXT.AlarmWarnUnAck := FALSE;
   STATUS[478].EXT.AckRequired := FALSE;
   STATUS[478].EXT.Maintanence := FALSE;
   STATUS[478].EXT.Operation := FALSE;
   STATUS[478].EXT.Forced := FALSE;
   STATUS[478].EXT.BIT29 := FALSE;
   STATUS[478].EXT.BIT30 := FALSE;
   STATUS[478].EXT.BIT31 := FALSE;
   STATUS[478].EXT.ModeBit1 := FALSE;
   STATUS[478].EXT.ModeBit2 := FALSE;
   STATUS[478].EXT.ModeBit3 := FALSE;
   STATUS[478].EXT.BIT19 := FALSE;
   STATUS[478].EXT.BIT20 := FALSE;
   STATUS[478].EXT.AlarmSuppressed := FALSE;
   STATUS[478].EXT.AlarmPresent := FALSE;
   STATUS[478].EXT.AlarmFailUnAck := FALSE;
   STATUS[478].Status := 0;
   STATUS[478].TimeStamp := 16#0000;
   STATUS[479].EXT.AlarmWarnUnAck := FALSE;
   STATUS[479].EXT.AckRequired := FALSE;
   STATUS[479].EXT.Maintanence := FALSE;
   STATUS[479].EXT.Operation := FALSE;
   STATUS[479].EXT.Forced := FALSE;
   STATUS[479].EXT.BIT29 := FALSE;
   STATUS[479].EXT.BIT30 := FALSE;
   STATUS[479].EXT.BIT31 := FALSE;
   STATUS[479].EXT.ModeBit1 := FALSE;
   STATUS[479].EXT.ModeBit2 := FALSE;
   STATUS[479].EXT.ModeBit3 := FALSE;
   STATUS[479].EXT.BIT19 := FALSE;
   STATUS[479].EXT.BIT20 := FALSE;
   STATUS[479].EXT.AlarmSuppressed := FALSE;
   STATUS[479].EXT.AlarmPresent := FALSE;
   STATUS[479].EXT.AlarmFailUnAck := FALSE;
   STATUS[479].Status := 0;
   STATUS[479].TimeStamp := 16#0000;
   STATUS[480].EXT.AlarmWarnUnAck := FALSE;
   STATUS[480].EXT.AckRequired := FALSE;
   STATUS[480].EXT.Maintanence := FALSE;
   STATUS[480].EXT.Operation := FALSE;
   STATUS[480].EXT.Forced := FALSE;
   STATUS[480].EXT.BIT29 := FALSE;
   STATUS[480].EXT.BIT30 := FALSE;
   STATUS[480].EXT.BIT31 := FALSE;
   STATUS[480].EXT.ModeBit1 := FALSE;
   STATUS[480].EXT.ModeBit2 := FALSE;
   STATUS[480].EXT.ModeBit3 := FALSE;
   STATUS[480].EXT.BIT19 := FALSE;
   STATUS[480].EXT.BIT20 := FALSE;
   STATUS[480].EXT.AlarmSuppressed := FALSE;
   STATUS[480].EXT.AlarmPresent := FALSE;
   STATUS[480].EXT.AlarmFailUnAck := FALSE;
   STATUS[480].Status := 0;
   STATUS[480].TimeStamp := 16#0000;
   STATUS[481].EXT.AlarmWarnUnAck := FALSE;
   STATUS[481].EXT.AckRequired := FALSE;
   STATUS[481].EXT.Maintanence := FALSE;
   STATUS[481].EXT.Operation := FALSE;
   STATUS[481].EXT.Forced := FALSE;
   STATUS[481].EXT.BIT29 := FALSE;
   STATUS[481].EXT.BIT30 := FALSE;
   STATUS[481].EXT.BIT31 := FALSE;
   STATUS[481].EXT.ModeBit1 := FALSE;
   STATUS[481].EXT.ModeBit2 := FALSE;
   STATUS[481].EXT.ModeBit3 := FALSE;
   STATUS[481].EXT.BIT19 := FALSE;
   STATUS[481].EXT.BIT20 := FALSE;
   STATUS[481].EXT.AlarmSuppressed := FALSE;
   STATUS[481].EXT.AlarmPresent := FALSE;
   STATUS[481].EXT.AlarmFailUnAck := FALSE;
   STATUS[481].Status := 0;
   STATUS[481].TimeStamp := 16#0000;
   STATUS[482].EXT.AlarmWarnUnAck := FALSE;
   STATUS[482].EXT.AckRequired := FALSE;
   STATUS[482].EXT.Maintanence := FALSE;
   STATUS[482].EXT.Operation := FALSE;
   STATUS[482].EXT.Forced := FALSE;
   STATUS[482].EXT.BIT29 := FALSE;
   STATUS[482].EXT.BIT30 := FALSE;
   STATUS[482].EXT.BIT31 := FALSE;
   STATUS[482].EXT.ModeBit1 := FALSE;
   STATUS[482].EXT.ModeBit2 := FALSE;
   STATUS[482].EXT.ModeBit3 := FALSE;
   STATUS[482].EXT.BIT19 := FALSE;
   STATUS[482].EXT.BIT20 := FALSE;
   STATUS[482].EXT.AlarmSuppressed := FALSE;
   STATUS[482].EXT.AlarmPresent := FALSE;
   STATUS[482].EXT.AlarmFailUnAck := FALSE;
   STATUS[482].Status := 0;
   STATUS[482].TimeStamp := 16#0000;
   STATUS[483].EXT.AlarmWarnUnAck := FALSE;
   STATUS[483].EXT.AckRequired := FALSE;
   STATUS[483].EXT.Maintanence := FALSE;
   STATUS[483].EXT.Operation := FALSE;
   STATUS[483].EXT.Forced := FALSE;
   STATUS[483].EXT.BIT29 := FALSE;
   STATUS[483].EXT.BIT30 := FALSE;
   STATUS[483].EXT.BIT31 := FALSE;
   STATUS[483].EXT.ModeBit1 := FALSE;
   STATUS[483].EXT.ModeBit2 := FALSE;
   STATUS[483].EXT.ModeBit3 := FALSE;
   STATUS[483].EXT.BIT19 := FALSE;
   STATUS[483].EXT.BIT20 := FALSE;
   STATUS[483].EXT.AlarmSuppressed := FALSE;
   STATUS[483].EXT.AlarmPresent := FALSE;
   STATUS[483].EXT.AlarmFailUnAck := FALSE;
   STATUS[483].Status := 0;
   STATUS[483].TimeStamp := 16#0000;
   STATUS[484].EXT.AlarmWarnUnAck := FALSE;
   STATUS[484].EXT.AckRequired := FALSE;
   STATUS[484].EXT.Maintanence := FALSE;
   STATUS[484].EXT.Operation := FALSE;
   STATUS[484].EXT.Forced := FALSE;
   STATUS[484].EXT.BIT29 := FALSE;
   STATUS[484].EXT.BIT30 := FALSE;
   STATUS[484].EXT.BIT31 := FALSE;
   STATUS[484].EXT.ModeBit1 := FALSE;
   STATUS[484].EXT.ModeBit2 := FALSE;
   STATUS[484].EXT.ModeBit3 := FALSE;
   STATUS[484].EXT.BIT19 := FALSE;
   STATUS[484].EXT.BIT20 := FALSE;
   STATUS[484].EXT.AlarmSuppressed := FALSE;
   STATUS[484].EXT.AlarmPresent := FALSE;
   STATUS[484].EXT.AlarmFailUnAck := FALSE;
   STATUS[484].Status := 0;
   STATUS[484].TimeStamp := 16#0000;
   STATUS[485].EXT.AlarmWarnUnAck := FALSE;
   STATUS[485].EXT.AckRequired := FALSE;
   STATUS[485].EXT.Maintanence := FALSE;
   STATUS[485].EXT.Operation := FALSE;
   STATUS[485].EXT.Forced := FALSE;
   STATUS[485].EXT.BIT29 := FALSE;
   STATUS[485].EXT.BIT30 := FALSE;
   STATUS[485].EXT.BIT31 := FALSE;
   STATUS[485].EXT.ModeBit1 := FALSE;
   STATUS[485].EXT.ModeBit2 := FALSE;
   STATUS[485].EXT.ModeBit3 := FALSE;
   STATUS[485].EXT.BIT19 := FALSE;
   STATUS[485].EXT.BIT20 := FALSE;
   STATUS[485].EXT.AlarmSuppressed := FALSE;
   STATUS[485].EXT.AlarmPresent := FALSE;
   STATUS[485].EXT.AlarmFailUnAck := FALSE;
   STATUS[485].Status := 0;
   STATUS[485].TimeStamp := 16#0000;
   STATUS[486].EXT.AlarmWarnUnAck := FALSE;
   STATUS[486].EXT.AckRequired := FALSE;
   STATUS[486].EXT.Maintanence := FALSE;
   STATUS[486].EXT.Operation := FALSE;
   STATUS[486].EXT.Forced := FALSE;
   STATUS[486].EXT.BIT29 := FALSE;
   STATUS[486].EXT.BIT30 := FALSE;
   STATUS[486].EXT.BIT31 := FALSE;
   STATUS[486].EXT.ModeBit1 := FALSE;
   STATUS[486].EXT.ModeBit2 := FALSE;
   STATUS[486].EXT.ModeBit3 := FALSE;
   STATUS[486].EXT.BIT19 := FALSE;
   STATUS[486].EXT.BIT20 := FALSE;
   STATUS[486].EXT.AlarmSuppressed := FALSE;
   STATUS[486].EXT.AlarmPresent := FALSE;
   STATUS[486].EXT.AlarmFailUnAck := FALSE;
   STATUS[486].Status := 0;
   STATUS[486].TimeStamp := 16#0000;
   STATUS[487].EXT.AlarmWarnUnAck := FALSE;
   STATUS[487].EXT.AckRequired := FALSE;
   STATUS[487].EXT.Maintanence := FALSE;
   STATUS[487].EXT.Operation := FALSE;
   STATUS[487].EXT.Forced := FALSE;
   STATUS[487].EXT.BIT29 := FALSE;
   STATUS[487].EXT.BIT30 := FALSE;
   STATUS[487].EXT.BIT31 := FALSE;
   STATUS[487].EXT.ModeBit1 := FALSE;
   STATUS[487].EXT.ModeBit2 := FALSE;
   STATUS[487].EXT.ModeBit3 := FALSE;
   STATUS[487].EXT.BIT19 := FALSE;
   STATUS[487].EXT.BIT20 := FALSE;
   STATUS[487].EXT.AlarmSuppressed := FALSE;
   STATUS[487].EXT.AlarmPresent := FALSE;
   STATUS[487].EXT.AlarmFailUnAck := FALSE;
   STATUS[487].Status := 0;
   STATUS[487].TimeStamp := 16#0000;
   STATUS[488].EXT.AlarmWarnUnAck := FALSE;
   STATUS[488].EXT.AckRequired := FALSE;
   STATUS[488].EXT.Maintanence := FALSE;
   STATUS[488].EXT.Operation := FALSE;
   STATUS[488].EXT.Forced := FALSE;
   STATUS[488].EXT.BIT29 := FALSE;
   STATUS[488].EXT.BIT30 := FALSE;
   STATUS[488].EXT.BIT31 := FALSE;
   STATUS[488].EXT.ModeBit1 := FALSE;
   STATUS[488].EXT.ModeBit2 := FALSE;
   STATUS[488].EXT.ModeBit3 := FALSE;
   STATUS[488].EXT.BIT19 := FALSE;
   STATUS[488].EXT.BIT20 := FALSE;
   STATUS[488].EXT.AlarmSuppressed := FALSE;
   STATUS[488].EXT.AlarmPresent := FALSE;
   STATUS[488].EXT.AlarmFailUnAck := FALSE;
   STATUS[488].Status := 0;
   STATUS[488].TimeStamp := 16#0000;
   STATUS[489].EXT.AlarmWarnUnAck := FALSE;
   STATUS[489].EXT.AckRequired := FALSE;
   STATUS[489].EXT.Maintanence := FALSE;
   STATUS[489].EXT.Operation := FALSE;
   STATUS[489].EXT.Forced := FALSE;
   STATUS[489].EXT.BIT29 := FALSE;
   STATUS[489].EXT.BIT30 := FALSE;
   STATUS[489].EXT.BIT31 := FALSE;
   STATUS[489].EXT.ModeBit1 := FALSE;
   STATUS[489].EXT.ModeBit2 := FALSE;
   STATUS[489].EXT.ModeBit3 := FALSE;
   STATUS[489].EXT.BIT19 := FALSE;
   STATUS[489].EXT.BIT20 := FALSE;
   STATUS[489].EXT.AlarmSuppressed := FALSE;
   STATUS[489].EXT.AlarmPresent := FALSE;
   STATUS[489].EXT.AlarmFailUnAck := FALSE;
   STATUS[489].Status := 0;
   STATUS[489].TimeStamp := 16#0000;
   STATUS[490].EXT.AlarmWarnUnAck := FALSE;
   STATUS[490].EXT.AckRequired := FALSE;
   STATUS[490].EXT.Maintanence := FALSE;
   STATUS[490].EXT.Operation := FALSE;
   STATUS[490].EXT.Forced := FALSE;
   STATUS[490].EXT.BIT29 := FALSE;
   STATUS[490].EXT.BIT30 := FALSE;
   STATUS[490].EXT.BIT31 := FALSE;
   STATUS[490].EXT.ModeBit1 := FALSE;
   STATUS[490].EXT.ModeBit2 := FALSE;
   STATUS[490].EXT.ModeBit3 := FALSE;
   STATUS[490].EXT.BIT19 := FALSE;
   STATUS[490].EXT.BIT20 := FALSE;
   STATUS[490].EXT.AlarmSuppressed := FALSE;
   STATUS[490].EXT.AlarmPresent := FALSE;
   STATUS[490].EXT.AlarmFailUnAck := FALSE;
   STATUS[490].Status := 0;
   STATUS[490].TimeStamp := 16#0000;
   STATUS[491].EXT.AlarmWarnUnAck := FALSE;
   STATUS[491].EXT.AckRequired := FALSE;
   STATUS[491].EXT.Maintanence := FALSE;
   STATUS[491].EXT.Operation := FALSE;
   STATUS[491].EXT.Forced := FALSE;
   STATUS[491].EXT.BIT29 := FALSE;
   STATUS[491].EXT.BIT30 := FALSE;
   STATUS[491].EXT.BIT31 := FALSE;
   STATUS[491].EXT.ModeBit1 := FALSE;
   STATUS[491].EXT.ModeBit2 := FALSE;
   STATUS[491].EXT.ModeBit3 := FALSE;
   STATUS[491].EXT.BIT19 := FALSE;
   STATUS[491].EXT.BIT20 := FALSE;
   STATUS[491].EXT.AlarmSuppressed := FALSE;
   STATUS[491].EXT.AlarmPresent := FALSE;
   STATUS[491].EXT.AlarmFailUnAck := FALSE;
   STATUS[491].Status := 0;
   STATUS[491].TimeStamp := 16#0000;
   STATUS[492].EXT.AlarmWarnUnAck := FALSE;
   STATUS[492].EXT.AckRequired := FALSE;
   STATUS[492].EXT.Maintanence := FALSE;
   STATUS[492].EXT.Operation := FALSE;
   STATUS[492].EXT.Forced := FALSE;
   STATUS[492].EXT.BIT29 := FALSE;
   STATUS[492].EXT.BIT30 := FALSE;
   STATUS[492].EXT.BIT31 := FALSE;
   STATUS[492].EXT.ModeBit1 := FALSE;
   STATUS[492].EXT.ModeBit2 := FALSE;
   STATUS[492].EXT.ModeBit3 := FALSE;
   STATUS[492].EXT.BIT19 := FALSE;
   STATUS[492].EXT.BIT20 := FALSE;
   STATUS[492].EXT.AlarmSuppressed := FALSE;
   STATUS[492].EXT.AlarmPresent := FALSE;
   STATUS[492].EXT.AlarmFailUnAck := FALSE;
   STATUS[492].Status := 0;
   STATUS[492].TimeStamp := 16#0000;
   STATUS[493].EXT.AlarmWarnUnAck := FALSE;
   STATUS[493].EXT.AckRequired := FALSE;
   STATUS[493].EXT.Maintanence := FALSE;
   STATUS[493].EXT.Operation := FALSE;
   STATUS[493].EXT.Forced := FALSE;
   STATUS[493].EXT.BIT29 := FALSE;
   STATUS[493].EXT.BIT30 := FALSE;
   STATUS[493].EXT.BIT31 := FALSE;
   STATUS[493].EXT.ModeBit1 := FALSE;
   STATUS[493].EXT.ModeBit2 := FALSE;
   STATUS[493].EXT.ModeBit3 := FALSE;
   STATUS[493].EXT.BIT19 := FALSE;
   STATUS[493].EXT.BIT20 := FALSE;
   STATUS[493].EXT.AlarmSuppressed := FALSE;
   STATUS[493].EXT.AlarmPresent := FALSE;
   STATUS[493].EXT.AlarmFailUnAck := FALSE;
   STATUS[493].Status := 0;
   STATUS[493].TimeStamp := 16#0000;
   STATUS[494].EXT.AlarmWarnUnAck := FALSE;
   STATUS[494].EXT.AckRequired := FALSE;
   STATUS[494].EXT.Maintanence := FALSE;
   STATUS[494].EXT.Operation := FALSE;
   STATUS[494].EXT.Forced := FALSE;
   STATUS[494].EXT.BIT29 := FALSE;
   STATUS[494].EXT.BIT30 := FALSE;
   STATUS[494].EXT.BIT31 := FALSE;
   STATUS[494].EXT.ModeBit1 := FALSE;
   STATUS[494].EXT.ModeBit2 := FALSE;
   STATUS[494].EXT.ModeBit3 := FALSE;
   STATUS[494].EXT.BIT19 := FALSE;
   STATUS[494].EXT.BIT20 := FALSE;
   STATUS[494].EXT.AlarmSuppressed := FALSE;
   STATUS[494].EXT.AlarmPresent := FALSE;
   STATUS[494].EXT.AlarmFailUnAck := FALSE;
   STATUS[494].Status := 0;
   STATUS[494].TimeStamp := 16#0000;
   STATUS[495].EXT.AlarmWarnUnAck := FALSE;
   STATUS[495].EXT.AckRequired := FALSE;
   STATUS[495].EXT.Maintanence := FALSE;
   STATUS[495].EXT.Operation := FALSE;
   STATUS[495].EXT.Forced := FALSE;
   STATUS[495].EXT.BIT29 := FALSE;
   STATUS[495].EXT.BIT30 := FALSE;
   STATUS[495].EXT.BIT31 := FALSE;
   STATUS[495].EXT.ModeBit1 := FALSE;
   STATUS[495].EXT.ModeBit2 := FALSE;
   STATUS[495].EXT.ModeBit3 := FALSE;
   STATUS[495].EXT.BIT19 := FALSE;
   STATUS[495].EXT.BIT20 := FALSE;
   STATUS[495].EXT.AlarmSuppressed := FALSE;
   STATUS[495].EXT.AlarmPresent := FALSE;
   STATUS[495].EXT.AlarmFailUnAck := FALSE;
   STATUS[495].Status := 0;
   STATUS[495].TimeStamp := 16#0000;
   STATUS[496].EXT.AlarmWarnUnAck := FALSE;
   STATUS[496].EXT.AckRequired := FALSE;
   STATUS[496].EXT.Maintanence := FALSE;
   STATUS[496].EXT.Operation := FALSE;
   STATUS[496].EXT.Forced := FALSE;
   STATUS[496].EXT.BIT29 := FALSE;
   STATUS[496].EXT.BIT30 := FALSE;
   STATUS[496].EXT.BIT31 := FALSE;
   STATUS[496].EXT.ModeBit1 := FALSE;
   STATUS[496].EXT.ModeBit2 := FALSE;
   STATUS[496].EXT.ModeBit3 := FALSE;
   STATUS[496].EXT.BIT19 := FALSE;
   STATUS[496].EXT.BIT20 := FALSE;
   STATUS[496].EXT.AlarmSuppressed := FALSE;
   STATUS[496].EXT.AlarmPresent := FALSE;
   STATUS[496].EXT.AlarmFailUnAck := FALSE;
   STATUS[496].Status := 0;
   STATUS[496].TimeStamp := 16#0000;
   STATUS[497].EXT.AlarmWarnUnAck := FALSE;
   STATUS[497].EXT.AckRequired := FALSE;
   STATUS[497].EXT.Maintanence := FALSE;
   STATUS[497].EXT.Operation := FALSE;
   STATUS[497].EXT.Forced := FALSE;
   STATUS[497].EXT.BIT29 := FALSE;
   STATUS[497].EXT.BIT30 := FALSE;
   STATUS[497].EXT.BIT31 := FALSE;
   STATUS[497].EXT.ModeBit1 := FALSE;
   STATUS[497].EXT.ModeBit2 := FALSE;
   STATUS[497].EXT.ModeBit3 := FALSE;
   STATUS[497].EXT.BIT19 := FALSE;
   STATUS[497].EXT.BIT20 := FALSE;
   STATUS[497].EXT.AlarmSuppressed := FALSE;
   STATUS[497].EXT.AlarmPresent := FALSE;
   STATUS[497].EXT.AlarmFailUnAck := FALSE;
   STATUS[497].Status := 0;
   STATUS[497].TimeStamp := 16#0000;
   STATUS[498].EXT.AlarmWarnUnAck := FALSE;
   STATUS[498].EXT.AckRequired := FALSE;
   STATUS[498].EXT.Maintanence := FALSE;
   STATUS[498].EXT.Operation := FALSE;
   STATUS[498].EXT.Forced := FALSE;
   STATUS[498].EXT.BIT29 := FALSE;
   STATUS[498].EXT.BIT30 := FALSE;
   STATUS[498].EXT.BIT31 := FALSE;
   STATUS[498].EXT.ModeBit1 := FALSE;
   STATUS[498].EXT.ModeBit2 := FALSE;
   STATUS[498].EXT.ModeBit3 := FALSE;
   STATUS[498].EXT.BIT19 := FALSE;
   STATUS[498].EXT.BIT20 := FALSE;
   STATUS[498].EXT.AlarmSuppressed := FALSE;
   STATUS[498].EXT.AlarmPresent := FALSE;
   STATUS[498].EXT.AlarmFailUnAck := FALSE;
   STATUS[498].Status := 0;
   STATUS[498].TimeStamp := 16#0000;
   STATUS[499].EXT.AlarmWarnUnAck := FALSE;
   STATUS[499].EXT.AckRequired := FALSE;
   STATUS[499].EXT.Maintanence := FALSE;
   STATUS[499].EXT.Operation := FALSE;
   STATUS[499].EXT.Forced := FALSE;
   STATUS[499].EXT.BIT29 := FALSE;
   STATUS[499].EXT.BIT30 := FALSE;
   STATUS[499].EXT.BIT31 := FALSE;
   STATUS[499].EXT.ModeBit1 := FALSE;
   STATUS[499].EXT.ModeBit2 := FALSE;
   STATUS[499].EXT.ModeBit3 := FALSE;
   STATUS[499].EXT.BIT19 := FALSE;
   STATUS[499].EXT.BIT20 := FALSE;
   STATUS[499].EXT.AlarmSuppressed := FALSE;
   STATUS[499].EXT.AlarmPresent := FALSE;
   STATUS[499].EXT.AlarmFailUnAck := FALSE;
   STATUS[499].Status := 0;
   STATUS[499].TimeStamp := 16#0000;
   STATUS[500].EXT.AlarmWarnUnAck := FALSE;
   STATUS[500].EXT.AckRequired := FALSE;
   STATUS[500].EXT.Maintanence := FALSE;
   STATUS[500].EXT.Operation := FALSE;
   STATUS[500].EXT.Forced := FALSE;
   STATUS[500].EXT.BIT29 := FALSE;
   STATUS[500].EXT.BIT30 := FALSE;
   STATUS[500].EXT.BIT31 := FALSE;
   STATUS[500].EXT.ModeBit1 := FALSE;
   STATUS[500].EXT.ModeBit2 := FALSE;
   STATUS[500].EXT.ModeBit3 := FALSE;
   STATUS[500].EXT.BIT19 := FALSE;
   STATUS[500].EXT.BIT20 := FALSE;
   STATUS[500].EXT.AlarmSuppressed := FALSE;
   STATUS[500].EXT.AlarmPresent := FALSE;
   STATUS[500].EXT.AlarmFailUnAck := FALSE;
   STATUS[500].Status := 0;
   STATUS[500].TimeStamp := 16#0000;
   STATUS[501].EXT.AlarmWarnUnAck := FALSE;
   STATUS[501].EXT.AckRequired := FALSE;
   STATUS[501].EXT.Maintanence := FALSE;
   STATUS[501].EXT.Operation := FALSE;
   STATUS[501].EXT.Forced := FALSE;
   STATUS[501].EXT.BIT29 := FALSE;
   STATUS[501].EXT.BIT30 := FALSE;
   STATUS[501].EXT.BIT31 := FALSE;
   STATUS[501].EXT.ModeBit1 := FALSE;
   STATUS[501].EXT.ModeBit2 := FALSE;
   STATUS[501].EXT.ModeBit3 := FALSE;
   STATUS[501].EXT.BIT19 := FALSE;
   STATUS[501].EXT.BIT20 := FALSE;
   STATUS[501].EXT.AlarmSuppressed := FALSE;
   STATUS[501].EXT.AlarmPresent := FALSE;
   STATUS[501].EXT.AlarmFailUnAck := FALSE;
   STATUS[501].Status := 0;
   STATUS[501].TimeStamp := 16#0000;
   STATUS[502].EXT.AlarmWarnUnAck := FALSE;
   STATUS[502].EXT.AckRequired := FALSE;
   STATUS[502].EXT.Maintanence := FALSE;
   STATUS[502].EXT.Operation := FALSE;
   STATUS[502].EXT.Forced := FALSE;
   STATUS[502].EXT.BIT29 := FALSE;
   STATUS[502].EXT.BIT30 := FALSE;
   STATUS[502].EXT.BIT31 := FALSE;
   STATUS[502].EXT.ModeBit1 := FALSE;
   STATUS[502].EXT.ModeBit2 := FALSE;
   STATUS[502].EXT.ModeBit3 := FALSE;
   STATUS[502].EXT.BIT19 := FALSE;
   STATUS[502].EXT.BIT20 := FALSE;
   STATUS[502].EXT.AlarmSuppressed := FALSE;
   STATUS[502].EXT.AlarmPresent := FALSE;
   STATUS[502].EXT.AlarmFailUnAck := FALSE;
   STATUS[502].Status := 0;
   STATUS[502].TimeStamp := 16#0000;
   STATUS[503].EXT.AlarmWarnUnAck := FALSE;
   STATUS[503].EXT.AckRequired := FALSE;
   STATUS[503].EXT.Maintanence := FALSE;
   STATUS[503].EXT.Operation := FALSE;
   STATUS[503].EXT.Forced := FALSE;
   STATUS[503].EXT.BIT29 := FALSE;
   STATUS[503].EXT.BIT30 := FALSE;
   STATUS[503].EXT.BIT31 := FALSE;
   STATUS[503].EXT.ModeBit1 := FALSE;
   STATUS[503].EXT.ModeBit2 := FALSE;
   STATUS[503].EXT.ModeBit3 := FALSE;
   STATUS[503].EXT.BIT19 := FALSE;
   STATUS[503].EXT.BIT20 := FALSE;
   STATUS[503].EXT.AlarmSuppressed := FALSE;
   STATUS[503].EXT.AlarmPresent := FALSE;
   STATUS[503].EXT.AlarmFailUnAck := FALSE;
   STATUS[503].Status := 0;
   STATUS[503].TimeStamp := 16#0000;
   STATUS[504].EXT.AlarmWarnUnAck := FALSE;
   STATUS[504].EXT.AckRequired := FALSE;
   STATUS[504].EXT.Maintanence := FALSE;
   STATUS[504].EXT.Operation := FALSE;
   STATUS[504].EXT.Forced := FALSE;
   STATUS[504].EXT.BIT29 := FALSE;
   STATUS[504].EXT.BIT30 := FALSE;
   STATUS[504].EXT.BIT31 := FALSE;
   STATUS[504].EXT.ModeBit1 := FALSE;
   STATUS[504].EXT.ModeBit2 := FALSE;
   STATUS[504].EXT.ModeBit3 := FALSE;
   STATUS[504].EXT.BIT19 := FALSE;
   STATUS[504].EXT.BIT20 := FALSE;
   STATUS[504].EXT.AlarmSuppressed := FALSE;
   STATUS[504].EXT.AlarmPresent := FALSE;
   STATUS[504].EXT.AlarmFailUnAck := FALSE;
   STATUS[504].Status := 0;
   STATUS[504].TimeStamp := 16#0000;
   STATUS[505].EXT.AlarmWarnUnAck := FALSE;
   STATUS[505].EXT.AckRequired := FALSE;
   STATUS[505].EXT.Maintanence := FALSE;
   STATUS[505].EXT.Operation := FALSE;
   STATUS[505].EXT.Forced := FALSE;
   STATUS[505].EXT.BIT29 := FALSE;
   STATUS[505].EXT.BIT30 := FALSE;
   STATUS[505].EXT.BIT31 := FALSE;
   STATUS[505].EXT.ModeBit1 := FALSE;
   STATUS[505].EXT.ModeBit2 := FALSE;
   STATUS[505].EXT.ModeBit3 := FALSE;
   STATUS[505].EXT.BIT19 := FALSE;
   STATUS[505].EXT.BIT20 := FALSE;
   STATUS[505].EXT.AlarmSuppressed := FALSE;
   STATUS[505].EXT.AlarmPresent := FALSE;
   STATUS[505].EXT.AlarmFailUnAck := FALSE;
   STATUS[505].Status := 0;
   STATUS[505].TimeStamp := 16#0000;
   STATUS[506].EXT.AlarmWarnUnAck := FALSE;
   STATUS[506].EXT.AckRequired := FALSE;
   STATUS[506].EXT.Maintanence := FALSE;
   STATUS[506].EXT.Operation := FALSE;
   STATUS[506].EXT.Forced := FALSE;
   STATUS[506].EXT.BIT29 := FALSE;
   STATUS[506].EXT.BIT30 := FALSE;
   STATUS[506].EXT.BIT31 := FALSE;
   STATUS[506].EXT.ModeBit1 := FALSE;
   STATUS[506].EXT.ModeBit2 := FALSE;
   STATUS[506].EXT.ModeBit3 := FALSE;
   STATUS[506].EXT.BIT19 := FALSE;
   STATUS[506].EXT.BIT20 := FALSE;
   STATUS[506].EXT.AlarmSuppressed := FALSE;
   STATUS[506].EXT.AlarmPresent := FALSE;
   STATUS[506].EXT.AlarmFailUnAck := FALSE;
   STATUS[506].Status := 0;
   STATUS[506].TimeStamp := 16#0000;
   STATUS[507].EXT.AlarmWarnUnAck := FALSE;
   STATUS[507].EXT.AckRequired := FALSE;
   STATUS[507].EXT.Maintanence := FALSE;
   STATUS[507].EXT.Operation := FALSE;
   STATUS[507].EXT.Forced := FALSE;
   STATUS[507].EXT.BIT29 := FALSE;
   STATUS[507].EXT.BIT30 := FALSE;
   STATUS[507].EXT.BIT31 := FALSE;
   STATUS[507].EXT.ModeBit1 := FALSE;
   STATUS[507].EXT.ModeBit2 := FALSE;
   STATUS[507].EXT.ModeBit3 := FALSE;
   STATUS[507].EXT.BIT19 := FALSE;
   STATUS[507].EXT.BIT20 := FALSE;
   STATUS[507].EXT.AlarmSuppressed := FALSE;
   STATUS[507].EXT.AlarmPresent := FALSE;
   STATUS[507].EXT.AlarmFailUnAck := FALSE;
   STATUS[507].Status := 0;
   STATUS[507].TimeStamp := 16#0000;
   STATUS[508].EXT.AlarmWarnUnAck := FALSE;
   STATUS[508].EXT.AckRequired := FALSE;
   STATUS[508].EXT.Maintanence := FALSE;
   STATUS[508].EXT.Operation := FALSE;
   STATUS[508].EXT.Forced := FALSE;
   STATUS[508].EXT.BIT29 := FALSE;
   STATUS[508].EXT.BIT30 := FALSE;
   STATUS[508].EXT.BIT31 := FALSE;
   STATUS[508].EXT.ModeBit1 := FALSE;
   STATUS[508].EXT.ModeBit2 := FALSE;
   STATUS[508].EXT.ModeBit3 := FALSE;
   STATUS[508].EXT.BIT19 := FALSE;
   STATUS[508].EXT.BIT20 := FALSE;
   STATUS[508].EXT.AlarmSuppressed := FALSE;
   STATUS[508].EXT.AlarmPresent := FALSE;
   STATUS[508].EXT.AlarmFailUnAck := FALSE;
   STATUS[508].Status := 0;
   STATUS[508].TimeStamp := 16#0000;
   STATUS[509].EXT.AlarmWarnUnAck := FALSE;
   STATUS[509].EXT.AckRequired := FALSE;
   STATUS[509].EXT.Maintanence := FALSE;
   STATUS[509].EXT.Operation := FALSE;
   STATUS[509].EXT.Forced := FALSE;
   STATUS[509].EXT.BIT29 := FALSE;
   STATUS[509].EXT.BIT30 := FALSE;
   STATUS[509].EXT.BIT31 := FALSE;
   STATUS[509].EXT.ModeBit1 := FALSE;
   STATUS[509].EXT.ModeBit2 := FALSE;
   STATUS[509].EXT.ModeBit3 := FALSE;
   STATUS[509].EXT.BIT19 := FALSE;
   STATUS[509].EXT.BIT20 := FALSE;
   STATUS[509].EXT.AlarmSuppressed := FALSE;
   STATUS[509].EXT.AlarmPresent := FALSE;
   STATUS[509].EXT.AlarmFailUnAck := FALSE;
   STATUS[509].Status := 0;
   STATUS[509].TimeStamp := 16#0000;
   STATUS[510].EXT.AlarmWarnUnAck := FALSE;
   STATUS[510].EXT.AckRequired := FALSE;
   STATUS[510].EXT.Maintanence := FALSE;
   STATUS[510].EXT.Operation := FALSE;
   STATUS[510].EXT.Forced := FALSE;
   STATUS[510].EXT.BIT29 := FALSE;
   STATUS[510].EXT.BIT30 := FALSE;
   STATUS[510].EXT.BIT31 := FALSE;
   STATUS[510].EXT.ModeBit1 := FALSE;
   STATUS[510].EXT.ModeBit2 := FALSE;
   STATUS[510].EXT.ModeBit3 := FALSE;
   STATUS[510].EXT.BIT19 := FALSE;
   STATUS[510].EXT.BIT20 := FALSE;
   STATUS[510].EXT.AlarmSuppressed := FALSE;
   STATUS[510].EXT.AlarmPresent := FALSE;
   STATUS[510].EXT.AlarmFailUnAck := FALSE;
   STATUS[510].Status := 0;
   STATUS[510].TimeStamp := 16#0000;
   STATUS[511].EXT.AlarmWarnUnAck := FALSE;
   STATUS[511].EXT.AckRequired := FALSE;
   STATUS[511].EXT.Maintanence := FALSE;
   STATUS[511].EXT.Operation := FALSE;
   STATUS[511].EXT.Forced := FALSE;
   STATUS[511].EXT.BIT29 := FALSE;
   STATUS[511].EXT.BIT30 := FALSE;
   STATUS[511].EXT.BIT31 := FALSE;
   STATUS[511].EXT.ModeBit1 := FALSE;
   STATUS[511].EXT.ModeBit2 := FALSE;
   STATUS[511].EXT.ModeBit3 := FALSE;
   STATUS[511].EXT.BIT19 := FALSE;
   STATUS[511].EXT.BIT20 := FALSE;
   STATUS[511].EXT.AlarmSuppressed := FALSE;
   STATUS[511].EXT.AlarmPresent := FALSE;
   STATUS[511].EXT.AlarmFailUnAck := FALSE;
   STATUS[511].Status := 0;
   STATUS[511].TimeStamp := 16#0000;
   STATUS[512].EXT.AlarmWarnUnAck := FALSE;
   STATUS[512].EXT.AckRequired := FALSE;
   STATUS[512].EXT.Maintanence := FALSE;
   STATUS[512].EXT.Operation := FALSE;
   STATUS[512].EXT.Forced := FALSE;
   STATUS[512].EXT.BIT29 := FALSE;
   STATUS[512].EXT.BIT30 := FALSE;
   STATUS[512].EXT.BIT31 := FALSE;
   STATUS[512].EXT.ModeBit1 := FALSE;
   STATUS[512].EXT.ModeBit2 := FALSE;
   STATUS[512].EXT.ModeBit3 := FALSE;
   STATUS[512].EXT.BIT19 := FALSE;
   STATUS[512].EXT.BIT20 := FALSE;
   STATUS[512].EXT.AlarmSuppressed := FALSE;
   STATUS[512].EXT.AlarmPresent := FALSE;
   STATUS[512].EXT.AlarmFailUnAck := FALSE;
   STATUS[512].Status := 0;
   STATUS[512].TimeStamp := 16#0000;
   STATUS[513].EXT.AlarmWarnUnAck := FALSE;
   STATUS[513].EXT.AckRequired := FALSE;
   STATUS[513].EXT.Maintanence := FALSE;
   STATUS[513].EXT.Operation := FALSE;
   STATUS[513].EXT.Forced := FALSE;
   STATUS[513].EXT.BIT29 := FALSE;
   STATUS[513].EXT.BIT30 := FALSE;
   STATUS[513].EXT.BIT31 := FALSE;
   STATUS[513].EXT.ModeBit1 := FALSE;
   STATUS[513].EXT.ModeBit2 := FALSE;
   STATUS[513].EXT.ModeBit3 := FALSE;
   STATUS[513].EXT.BIT19 := FALSE;
   STATUS[513].EXT.BIT20 := FALSE;
   STATUS[513].EXT.AlarmSuppressed := FALSE;
   STATUS[513].EXT.AlarmPresent := FALSE;
   STATUS[513].EXT.AlarmFailUnAck := FALSE;
   STATUS[513].Status := 0;
   STATUS[513].TimeStamp := 16#0000;
   STATUS[514].EXT.AlarmWarnUnAck := FALSE;
   STATUS[514].EXT.AckRequired := FALSE;
   STATUS[514].EXT.Maintanence := FALSE;
   STATUS[514].EXT.Operation := FALSE;
   STATUS[514].EXT.Forced := FALSE;
   STATUS[514].EXT.BIT29 := FALSE;
   STATUS[514].EXT.BIT30 := FALSE;
   STATUS[514].EXT.BIT31 := FALSE;
   STATUS[514].EXT.ModeBit1 := FALSE;
   STATUS[514].EXT.ModeBit2 := FALSE;
   STATUS[514].EXT.ModeBit3 := FALSE;
   STATUS[514].EXT.BIT19 := FALSE;
   STATUS[514].EXT.BIT20 := FALSE;
   STATUS[514].EXT.AlarmSuppressed := FALSE;
   STATUS[514].EXT.AlarmPresent := FALSE;
   STATUS[514].EXT.AlarmFailUnAck := FALSE;
   STATUS[514].Status := 0;
   STATUS[514].TimeStamp := 16#0000;
   STATUS[515].EXT.AlarmWarnUnAck := FALSE;
   STATUS[515].EXT.AckRequired := FALSE;
   STATUS[515].EXT.Maintanence := FALSE;
   STATUS[515].EXT.Operation := FALSE;
   STATUS[515].EXT.Forced := FALSE;
   STATUS[515].EXT.BIT29 := FALSE;
   STATUS[515].EXT.BIT30 := FALSE;
   STATUS[515].EXT.BIT31 := FALSE;
   STATUS[515].EXT.ModeBit1 := FALSE;
   STATUS[515].EXT.ModeBit2 := FALSE;
   STATUS[515].EXT.ModeBit3 := FALSE;
   STATUS[515].EXT.BIT19 := FALSE;
   STATUS[515].EXT.BIT20 := FALSE;
   STATUS[515].EXT.AlarmSuppressed := FALSE;
   STATUS[515].EXT.AlarmPresent := FALSE;
   STATUS[515].EXT.AlarmFailUnAck := FALSE;
   STATUS[515].Status := 0;
   STATUS[515].TimeStamp := 16#0000;
   STATUS[516].EXT.AlarmWarnUnAck := FALSE;
   STATUS[516].EXT.AckRequired := FALSE;
   STATUS[516].EXT.Maintanence := FALSE;
   STATUS[516].EXT.Operation := FALSE;
   STATUS[516].EXT.Forced := FALSE;
   STATUS[516].EXT.BIT29 := FALSE;
   STATUS[516].EXT.BIT30 := FALSE;
   STATUS[516].EXT.BIT31 := FALSE;
   STATUS[516].EXT.ModeBit1 := FALSE;
   STATUS[516].EXT.ModeBit2 := FALSE;
   STATUS[516].EXT.ModeBit3 := FALSE;
   STATUS[516].EXT.BIT19 := FALSE;
   STATUS[516].EXT.BIT20 := FALSE;
   STATUS[516].EXT.AlarmSuppressed := FALSE;
   STATUS[516].EXT.AlarmPresent := FALSE;
   STATUS[516].EXT.AlarmFailUnAck := FALSE;
   STATUS[516].Status := 0;
   STATUS[516].TimeStamp := 16#0000;
   STATUS[517].EXT.AlarmWarnUnAck := FALSE;
   STATUS[517].EXT.AckRequired := FALSE;
   STATUS[517].EXT.Maintanence := FALSE;
   STATUS[517].EXT.Operation := FALSE;
   STATUS[517].EXT.Forced := FALSE;
   STATUS[517].EXT.BIT29 := FALSE;
   STATUS[517].EXT.BIT30 := FALSE;
   STATUS[517].EXT.BIT31 := FALSE;
   STATUS[517].EXT.ModeBit1 := FALSE;
   STATUS[517].EXT.ModeBit2 := FALSE;
   STATUS[517].EXT.ModeBit3 := FALSE;
   STATUS[517].EXT.BIT19 := FALSE;
   STATUS[517].EXT.BIT20 := FALSE;
   STATUS[517].EXT.AlarmSuppressed := FALSE;
   STATUS[517].EXT.AlarmPresent := FALSE;
   STATUS[517].EXT.AlarmFailUnAck := FALSE;
   STATUS[517].Status := 0;
   STATUS[517].TimeStamp := 16#0000;
   STATUS[518].EXT.AlarmWarnUnAck := FALSE;
   STATUS[518].EXT.AckRequired := FALSE;
   STATUS[518].EXT.Maintanence := FALSE;
   STATUS[518].EXT.Operation := FALSE;
   STATUS[518].EXT.Forced := FALSE;
   STATUS[518].EXT.BIT29 := FALSE;
   STATUS[518].EXT.BIT30 := FALSE;
   STATUS[518].EXT.BIT31 := FALSE;
   STATUS[518].EXT.ModeBit1 := FALSE;
   STATUS[518].EXT.ModeBit2 := FALSE;
   STATUS[518].EXT.ModeBit3 := FALSE;
   STATUS[518].EXT.BIT19 := FALSE;
   STATUS[518].EXT.BIT20 := FALSE;
   STATUS[518].EXT.AlarmSuppressed := FALSE;
   STATUS[518].EXT.AlarmPresent := FALSE;
   STATUS[518].EXT.AlarmFailUnAck := FALSE;
   STATUS[518].Status := 0;
   STATUS[518].TimeStamp := 16#0000;
   STATUS[519].EXT.AlarmWarnUnAck := FALSE;
   STATUS[519].EXT.AckRequired := FALSE;
   STATUS[519].EXT.Maintanence := FALSE;
   STATUS[519].EXT.Operation := FALSE;
   STATUS[519].EXT.Forced := FALSE;
   STATUS[519].EXT.BIT29 := FALSE;
   STATUS[519].EXT.BIT30 := FALSE;
   STATUS[519].EXT.BIT31 := FALSE;
   STATUS[519].EXT.ModeBit1 := FALSE;
   STATUS[519].EXT.ModeBit2 := FALSE;
   STATUS[519].EXT.ModeBit3 := FALSE;
   STATUS[519].EXT.BIT19 := FALSE;
   STATUS[519].EXT.BIT20 := FALSE;
   STATUS[519].EXT.AlarmSuppressed := FALSE;
   STATUS[519].EXT.AlarmPresent := FALSE;
   STATUS[519].EXT.AlarmFailUnAck := FALSE;
   STATUS[519].Status := 0;
   STATUS[519].TimeStamp := 16#0000;
   STATUS[520].EXT.AlarmWarnUnAck := FALSE;
   STATUS[520].EXT.AckRequired := FALSE;
   STATUS[520].EXT.Maintanence := FALSE;
   STATUS[520].EXT.Operation := FALSE;
   STATUS[520].EXT.Forced := FALSE;
   STATUS[520].EXT.BIT29 := FALSE;
   STATUS[520].EXT.BIT30 := FALSE;
   STATUS[520].EXT.BIT31 := FALSE;
   STATUS[520].EXT.ModeBit1 := FALSE;
   STATUS[520].EXT.ModeBit2 := FALSE;
   STATUS[520].EXT.ModeBit3 := FALSE;
   STATUS[520].EXT.BIT19 := FALSE;
   STATUS[520].EXT.BIT20 := FALSE;
   STATUS[520].EXT.AlarmSuppressed := FALSE;
   STATUS[520].EXT.AlarmPresent := FALSE;
   STATUS[520].EXT.AlarmFailUnAck := FALSE;
   STATUS[520].Status := 0;
   STATUS[520].TimeStamp := 16#0000;
   STATUS[521].EXT.AlarmWarnUnAck := FALSE;
   STATUS[521].EXT.AckRequired := FALSE;
   STATUS[521].EXT.Maintanence := FALSE;
   STATUS[521].EXT.Operation := FALSE;
   STATUS[521].EXT.Forced := FALSE;
   STATUS[521].EXT.BIT29 := FALSE;
   STATUS[521].EXT.BIT30 := FALSE;
   STATUS[521].EXT.BIT31 := FALSE;
   STATUS[521].EXT.ModeBit1 := FALSE;
   STATUS[521].EXT.ModeBit2 := FALSE;
   STATUS[521].EXT.ModeBit3 := FALSE;
   STATUS[521].EXT.BIT19 := FALSE;
   STATUS[521].EXT.BIT20 := FALSE;
   STATUS[521].EXT.AlarmSuppressed := FALSE;
   STATUS[521].EXT.AlarmPresent := FALSE;
